// TwinCAT 3 PLC project TE1096_04
// Title: TE1096-04-SISS
// Company: Tegan Innovations Ltd.
// Author: oldschoo1
// ProjectVersion: 1.0.0
// Description: Stopper Insertion/Screw Station, 4th station of the EAGLE production line
// ProgramVersion: 3.1.4024.0
// libraries:
//   Tc2_EthernetIP, * (Beckhoff Automation GmbH)
//   Tc2_MC2, * (Beckhoff Automation GmbH)
//   Tc2_Standard, * (Beckhoff Automation GmbH)
//   Tc2_System, * (Beckhoff Automation GmbH)
//   Tc2_Utilities, * (Beckhoff Automation GmbH)
//   Tc3_Module, * (Beckhoff Automation GmbH)
// project tree:
//   DUTs/00_HMI/ ST_Chart.TcDUT, StPoint.TcDUT, ST_UserLogHMI.TcDUT
//   DUTs/01_MASTER/ E_MachineState.TcDUT, ST_ActiveEventsHMI.TcDUT, ST_AlarmHistory.TcDUT, ST_Events.TcDUT, ST_MachineStatus.TcDUT, ST_MasterCTRL.TcDUT, ST_ModuleCMD.TcDUT, ST_ModuleStatus.TcDUT, ST_SafetyPLC.TcDUT
//   DUTs/02_Y_AXIS/ E_AxisErrorID.TcDUT, E_AxisState.TcDUT, ST_Y_Axis.TcDUT
//   DUTs/03_KISTLER/ E_KistlerErrorID.TcDUT, E_KistlerState.TcDUT, ST_Kistler.TcDUT, ST_KistlerData_Temporary.TcDUT, ST_KistlerData_CMD.TcDUT, ST_KistlerData_Status.TcDUT
//   DUTs/04_SMAC/ E_SmacState.TcDUT, ST_Smac.TcDUT
//   DUTs/04_SMAC/FUNCTIONS/ ST_CYC_MAN.TcDUT, ST_Phasing_Home.TcDUT
//   DUTs/04_SMAC/I_O/ ST_SMAC_I_O.TcDUT
//   DUTs/05_ProcessCycle/ E_ProcessCycle.TcDUT, ST_ProcessReport.TcDUT
//   GVLs/ ETHIP.TcGVL, GVL_CONSTANTS.TcGVL, GVL_MODULES.TcGVL, GVL_PERSISTENT.TcGVL, GVL_HMI.TcGVL, GVL_IO.TcGVL, GVL_MASTER.TcGVL, GVL_UTILITIES.TcGVL
//   / PlcTask.TcTTO, PulseTask.TcTTO
//   POUs/00_MASTER/ D_FaultHandling.TcPOU, PRG_MasterSystemTime.TcPOU, A_Master.TcPOU, B_Safety.TcPOU, C_Machine_CTRL.TcPOU
//   POUs/01_MODULES/AXIS_Y/ PRG_Fault_Axis_Y.TcPOU, Y_Master_Y_Axis.TcPOU
//   POUs/01_MODULES/KISTLER/ K_Master_Kistler.TcPOU, PRG_Fault_Kistler.TcPOU
//   POUs/01_MODULES/SMAC/ PRG_Fault_SMAC.TcPOU, S_Master_SMAC.TcPOU
//   POUs/02_HMI/ A_HMI.TcPOU
//   POUs/03_Utilities/ FB_ArrayOfByte2Real.TcPOU, FB_BytesToReal.TcPOU, FB_Byte_To_Bits.TcPOU, FB_Chart.TcPOU, FB_DistanceMonitor.TcPOU, FB_EventLog.TcPOU, FB_ForceMonitor.TcPOU, FB_GripperCtrl.TcPOU, FB_Real2ArrayOfByte.TcPOU, FB_Scale.TcPOU, FB_TerminalInfo.TcPOU, FB_TimeControl.TcPOU, FUN_PackBoolArrayToByte.TcPOU, FB_UnpackByteToBoolArray.TcPOU, PRG_SysTime.TcPOU, FB_Pulse.TcPOU, PRG_SysPulses.TcPOU
//   POUs/03_Utilities/SMAC/ FB_ErrorReset.TcPOU, FB_SmacCycleMan.TcPOU, FB_SmacInitialization.TcPOU
//   POUs/ MAIN.TcPOU
// real-time tasks:
//   TASK PulseTask: cycle T#2ms, priority 5, ADS port 352
//   TASK PlcTask: cycle T#10ms, priority 20, ADS port 350
// motion (NC):
//   TASK NC-Task 1 SAF: cycle T#2ms, priority 4, ADS port 501
//   TASK NC-Task 1 SVB: cycle T#10ms, priority 8, ADS port 511
//   AXIS Y_Axis (id 1)
//     Dynamic: Acceleration=1231.5, Deceleration=1231.5, Jerk=3694.5
//     Velo: RefSearch=8.21, RefSync=8.21, SlowManual=41.05, FastManual=246.3, Fast=821, Maximum=821
//     MotionControl: Time=1
//     OtherSettings: AllowMotionCmdToSlave=true, DataPersistence=true
//     encoder EncType=19
//       EncPara: ScaleFactorNumerator=10, ScaleFactorDenominator=1048576, MaxCount=#xffffffff
//         SoftEndMinControl: Enable=true, Range=4.3
//         SoftEndMaxControl: Enable=true, Range=111
//     drive DrvType=16
//       DrvPara: MaxCount=#xffffffff, DriveControlDWord=#x00020000
//         Analog: VeloReferenz=903.1, VeloScale=32, TorqueSetpointScale=10, ScaleFactorActTorque=0.1
//         TimeComp: TaskDelayCycles=1
//     controller CtrType=1
//       CtrPara: PriorControlFactor=1
//         PosDiffControl: Range=1.3, Time=0.5
//         Observer: BandWidth=20
// I/O:
//   DEVICE EtherCAT Master (disabled), AmsNetId 192.168.0.127.2.1
//     Term 1 (EK1100) [EK1100 EtherCAT Coupler (2A E-Bus)]
//       Term 2 (EL6070-0033) [EL6070-0033 1Ch. Licence key terminal, individual licences]
//       Term 3 (EL6910) [EL6910, TwinSAFE PLC]
//       Term 4 (EL1918) [EL1918, 8Ch. Safety Input 24V, TwinSAFE]
//         modules: Module 1 (FSOE), Module 2 (FSLOGIC)
//       Term 5 (EL1918) [EL1918, 8Ch. Safety Input 24V, TwinSAFE]
//         modules: Module 1 (FSOE), Module 2 (FSLOGIC)
//       Term 6 (EL2904) [EL2904, 4 Ch. Safety Output 24V, 0.5A, TwinSAFE]
//         modules: Module 1 (FSOES), Module 2 (DO)
//       Term 7 (EL2904) [EL2904, 4 Ch. Safety Output 24V, 0.5A, TwinSAFE]
//         modules: Module 1 (FSOES), Module 2 (DO)
//       Term 8 (EL1809) [EL1809 16Ch. Dig. Input 24V, 3ms]
//       Term 9 (EL1809) [EL1809 16Ch. Dig. Input 24V, 3ms]
//       Term 10 (EL2809-0015) [EL2809-0015 16Ch. Dig. Output 24V DC, 0.35A, not short-circuit proof]
//       Term 11 (EL9576) [EL9576 Brake chopper terminal]
//       Term 12 (EL7211-0010) [EL7211-0010 1Ch. MDP742 Servo motor output stage with OCT (50V, 4.5A RMS)]
//       Term 14 (EL9011) [EL9011 End Terminal]
//     Box 13 (maXYmos) [5877A5847A]
//   DEVICE Device 2 (TC3 EIP Scanner), AmsNetId 192.168.0.127.3.1
//     VLC-2-EIP // <INFO> 192.168.7.180, VLC-2-EIP (ProdCode: 58072, Rev: 2.94, Mac: 00:03:19:45:01:01) </INFO> <EDS> C:\TwinCAT\3.1\Config\Io\EtherNetIP\VLC-2-EIP.eds </EDS>
// variable links:
//   NC-Task 1 SAF/Axes/Y_Axis <-> EtherCAT Master/Term 1 (EK1100)/Term 12 (EL7211-0010)
//     Drive/Inputs/In/nDcOutputTime <-> InfoData/DcOutputShift
//     Drive/Inputs/In/nState1 <-> DRV Statusword/Statusword
//     Drive/Inputs/In/nState2 <-> DRV Statusword/Statusword @bit 8
//     Drive/Inputs/In/nState4 @bit 1 <-> WcState/InputToggle
//     Drive/Inputs/In/nState4 <-> WcState/WcState
//     Drive/Outputs/Out/nCtrl1 <-> DRV Controlword/Controlword
//     Drive/Outputs/Out/nCtrl2 <-> DRV Controlword/Controlword @bit 8
//     Drive/Outputs/Out/nDataOut2 <-> DRV Target velocity/Target velocity
//     Enc/Inputs/In/nDataIn1 <-> FB Position/Position
//     Enc/Inputs/In/nDcInputTime <-> InfoData/DcInputShift
//     Enc/Inputs/In/nState4 @bit 1 <-> WcState/InputToggle
//     Enc/Inputs/In/nState4 <-> WcState/WcState
//   TE1096-04/TE1096-04 Instance <-> Device 2 (TC3 EIP Scanner)/VLC-2-EIP
//     PlcTask Inputs/GVL_MODULES.stSmacIO.inCurrentMacro <-> Connection 1 (Input/Output)/Inputs/I_MacroCallIndicator
//     PlcTask Inputs/GVL_MODULES.stSmacIO.inCurrentPositionLinear <-> Connection 1 (Input/Output)/Inputs/I_PositionActualVal_1
//     PlcTask Inputs/GVL_MODULES.stSmacIO.inCurrentPositionRotative <-> Connection 1 (Input/Output)/Inputs/I_PositionActualVal_2
//     PlcTask Inputs/GVL_MODULES.stSmacIO.inCurrentValueLinear <-> Connection 1 (Input/Output)/Inputs/I_CurrentVal_1
//     PlcTask Inputs/GVL_MODULES.stSmacIO.inCurrentValueRotative <-> Connection 1 (Input/Output)/Inputs/I_CurrentVal_2
//     PlcTask Inputs/GVL_MODULES.stSmacIO.inErrorIDLinear <-> Connection 1 (Input/Output)/Inputs/I_FollowingError_1
//     PlcTask Inputs/GVL_MODULES.stSmacIO.inErrorIDRotative <-> Connection 1 (Input/Output)/Inputs/I_FollowingError_2
//     PlcTask Inputs/GVL_MODULES.stSmacIO.inModeOfOperationLinear <-> Connection 1 (Input/Output)/Inputs/I_ModeofOperationDisplay_1
//     PlcTask Inputs/GVL_MODULES.stSmacIO.inModeOfOperationRotative <-> Connection 1 (Input/Output)/Inputs/I_ModeofOperationDisplay_2
//     PlcTask Inputs/GVL_MODULES.stSmacIO.inStatusWordLinear <-> Connection 1 (Input/Output)/Inputs/I_StatusWord_1
//     PlcTask Inputs/GVL_MODULES.stSmacIO.inStatusWordRotative <-> Connection 1 (Input/Output)/Inputs/I_StatusWord_2
//     PlcTask Outputs/GVL_MODULES.stSmacIO.qnControlWordLinear <-> Connection 1 (Input/Output)/Outputs/O_ControlWord_1
//     PlcTask Outputs/GVL_MODULES.stSmacIO.qnControlWordRotative <-> Connection 1 (Input/Output)/Outputs/O_ControlWord_2
//     PlcTask Outputs/GVL_MODULES.stSmacIO.qnModeOfOperationLinear <-> Connection 1 (Input/Output)/Outputs/O_ModesofOperation_1
//     PlcTask Outputs/GVL_MODULES.stSmacIO.qnModeOfOperationRotative <-> Connection 1 (Input/Output)/Outputs/O_ModesofOperation_2
//     PlcTask Outputs/GVL_MODULES.stSmacIO.qnSetAcceleraionLinear <-> Connection 1 (Input/Output)/Outputs/O_ProfileAcceleration_1
//     PlcTask Outputs/GVL_MODULES.stSmacIO.qnSetAcceleraionRotative <-> Connection 1 (Input/Output)/Outputs/O_ProfileAcceleration_2
//     PlcTask Outputs/GVL_MODULES.stSmacIO.qnSetMacroNumber <-> Connection 1 (Input/Output)/Outputs/O_MacroNumber
//     PlcTask Outputs/GVL_MODULES.stSmacIO.qnSetMaxiumTorqueLinear <-> Connection 1 (Input/Output)/Outputs/O_MaximumTorque_1
//     PlcTask Outputs/GVL_MODULES.stSmacIO.qnSetMaxiumTorqueRotative <-> Connection 1 (Input/Output)/Outputs/O_MaximumTorque_2
//     PlcTask Outputs/GVL_MODULES.stSmacIO.qnSetPointLinear <-> Connection 1 (Input/Output)/Outputs/O_Setpoint_1
//     PlcTask Outputs/GVL_MODULES.stSmacIO.qnSetPointRotative <-> Connection 1 (Input/Output)/Outputs/O_Setpoint_2
//     PlcTask Outputs/GVL_MODULES.stSmacIO.qnSetVelocityLinear <-> Connection 1 (Input/Output)/Outputs/O_ProfileVelocity_1
//     PlcTask Outputs/GVL_MODULES.stSmacIO.qnSetVelocityRotative <-> Connection 1 (Input/Output)/Outputs/O_ProfileVelocity_2
//   TE1096-04/TE1096-04 Instance <-> EtherCAT Master/Box 13 (maXYmos)
//     PlcTask Inputs/GVL_IO.iStatusBytes <-> Inputs0/1 Byte In (0)
//     PlcTask Inputs/GVL_IO.iStatusBytes @bit {8..1592 step 8} <-> Inputs0/1 Byte In ({1..199})  (199 links)
//     PlcTask Inputs/GVL_IO.nKistlermaXYmosState <-> InfoData/State
//     PlcTask Outputs/GVL_IO.qControlBytes <-> Outputs0/1 Byte Out (0)
//     PlcTask Outputs/GVL_IO.qControlBytes @bit {8..1592 step 8} <-> Outputs0/1 Byte Out ({1..199})  (199 links)
//   TE1096-04/TE1096-04 Instance <-> EtherCAT Master/Term 1 (EK1100)
//     PlcTask Inputs/GVL_IO.nEK1100State <-> InfoData/State
//   TE1096-04/TE1096-04 Instance <-> EtherCAT Master/Term 1 (EK1100)/Term 10 (EL2809-0015)
//     PlcTask Inputs/GVL_IO.nEL2809State <-> InfoData/State
//     PlcTask Outputs/GVL_IO.qCycleIndicator_GreenLED <-> Channel 8/Output
//     PlcTask Outputs/GVL_IO.qCycleIndicator_RedLED <-> Channel 7/Output
//     PlcTask Outputs/GVL_IO.qGripperA_Close <-> Channel 3/Output
//     PlcTask Outputs/GVL_IO.qGripperA_Open <-> Channel 4/Output
//     PlcTask Outputs/GVL_IO.qGripperB_Close <-> Channel 5/Output
//     PlcTask Outputs/GVL_IO.qGripperB_Open <-> Channel 6/Output
//     PlcTask Outputs/GVL_IO.qKistlerCTRL_Sig{1..4} <-> Channel {9..12}/Output  (4 links)
//     PlcTask Outputs/GVL_IO.qResetButton_LED <-> Channel 2/Output
//     PlcTask Outputs/GVL_IO.qSmacCTRL_Sig1 <-> Channel 13/Output
//     PlcTask Outputs/GVL_IO.qSmacCTRL_Sig2 <-> Channel 14/Output
//     PlcTask Outputs/GVL_IO.qSmacCTRL_Sig3 <-> Channel 15/Output
//     PlcTask Outputs/GVL_IO.qStartButton_LED <-> Channel 1/Output
//   TE1096-04/TE1096-04 Instance <-> EtherCAT Master/Term 1 (EK1100)/Term 11 (EL9576)
//     PlcTask Inputs/GVL_IO.nEL9576State <-> InfoData/State
//   TE1096-04/TE1096-04 Instance <-> EtherCAT Master/Term 1 (EK1100)/Term 12 (EL7211-0010)
//     PlcTask Inputs/GVL_IO.nEL7211State <-> InfoData/State
//   TE1096-04/TE1096-04 Instance <-> EtherCAT Master/Term 1 (EK1100)/Term 2 (EL6070-0033)
//     PlcTask Inputs/GVL_IO.nEL6070State <-> InfoData/State
//   TE1096-04/TE1096-04 Instance <-> EtherCAT Master/Term 1 (EK1100)/Term 3 (EL6910)
//     PlcTask Inputs/GVL_IO.isDoorClosed <-> StandardInputs/Standard Out Var 21
//     PlcTask Inputs/GVL_IO.isDoorLocked <-> StandardInputs/Standard Out Var 23
//     PlcTask Inputs/GVL_IO.isEStop_OK <-> StandardInputs/Standard Out Var 20
//     PlcTask Inputs/GVL_IO.isLightBeam_NotCrossed <-> StandardInputs/Standard Out Var 25
//     PlcTask Inputs/GVL_IO.isLightBeam_OK <-> StandardInputs/Standard Out Var 26
//     PlcTask Inputs/GVL_IO.isSafetyCom_Error <-> StandardInputs/Standard Out Var 19
//     PlcTask Inputs/GVL_IO.isSafetyFB_Error <-> StandardInputs/Standard Out Var 18
//     PlcTask Inputs/GVL_IO.isSafetyRunning <-> StandardInputs/Standard Out Var 17
//     PlcTask Inputs/GVL_IO.isSafety_OK <-> StandardInputs/Standard Out Var 30
//     PlcTask Inputs/GVL_IO.isTwoHands_SIGNAL <-> StandardInputs/Standard Out Var 28
//     PlcTask Inputs/GVL_IO.nEL6910State <-> InfoData/State
//     PlcTask Outputs/GVL_IO.qsLightBeam_MutingActive <-> StandardOutputs/Standard In Var 24
//     PlcTask Outputs/GVL_IO.qsLockDoorCMD <-> StandardOutputs/Standard In Var 22
//     PlcTask Outputs/GVL_IO.qsSafetyErrorAck <-> StandardOutputs/Standard In Var 1
//     PlcTask Outputs/GVL_IO.qsSafetyRun <-> StandardOutputs/Standard In Var 3
//     PlcTask Outputs/GVL_IO.qsTwoHandsMonitoring <-> StandardOutputs/Standard In Var 27
//   TE1096-04/TE1096-04 Instance <-> EtherCAT Master/Term 1 (EK1100)/Term 4 (EL1918)
//     PlcTask Inputs/GVL_IO.iDoorInterlock_Ch1 <-> Module 1 (FSOE)/FSoE Inputs/FSOE/FSIN Module 4.Input
//     PlcTask Inputs/GVL_IO.iDoorInterlock_Ch2 <-> Module 1 (FSOE)/FSoE Inputs/FSOE/FSIN Module 5.Input
//     PlcTask Inputs/GVL_IO.iDoorInterlock_FB <-> Module 1 (FSOE)/FSoE Inputs/FSOE/FSIN Module 6.Input
//     PlcTask Inputs/GVL_IO.iE_Stop_Ch1 <-> Module 1 (FSOE)/FSoE Inputs/FSOE/FSIN Module 1.Input
//     PlcTask Inputs/GVL_IO.iE_Stop_Ch2 <-> Module 1 (FSOE)/FSoE Inputs/FSOE/FSIN Module 2.Input
//     PlcTask Inputs/GVL_IO.iIndraDrive_Contactor_FB <-> Module 1 (FSOE)/FSoE Inputs/FSOE/FSIN Module 7.Input
//     PlcTask Inputs/GVL_IO.iResetButton <-> Module 1 (FSOE)/FSoE Inputs/FSOE/FSIN Module 3.Input
//     PlcTask Inputs/GVL_IO.iSmacSTO_FB <-> Module 1 (FSOE)/FSoE Inputs/FSOE/FSIN Module 8.Input
//     PlcTask Inputs/GVL_IO.nEL1918_1State <-> InfoData/State
//   TE1096-04/TE1096-04 Instance <-> EtherCAT Master/Term 1 (EK1100)/Term 5 (EL1918)
//     PlcTask Inputs/GVL_IO.iAxis_1_SafetyRelayFB <-> Module 1 (FSOE)/FSoE Inputs/FSOE/FSIN Module 6.Input
//     PlcTask Inputs/GVL_IO.iPilz2_FB <-> Module 1 (FSOE)/FSoE Inputs/FSOE/FSIN Module 5.Input
//     PlcTask Inputs/GVL_IO.iSafetyBeam_Signal <-> Module 1 (FSOE)/FSoE Inputs/FSOE/FSIN Module 7.Input
//     PlcTask Inputs/GVL_IO.iTouchBtn_1_NC <-> Module 1 (FSOE)/FSoE Inputs/FSOE/FSIN Module 1.Input
//     PlcTask Inputs/GVL_IO.iTouchBtn_2_NC <-> Module 1 (FSOE)/FSoE Inputs/FSOE/FSIN Module 2.Input
//     PlcTask Inputs/GVL_IO.iTouchBtn_1_NO <-> Module 1 (FSOE)/FSoE Inputs/FSOE/FSIN Module 3.Input
//     PlcTask Inputs/GVL_IO.iTouchBtn_2_NO <-> Module 1 (FSOE)/FSoE Inputs/FSOE/FSIN Module 4.Input
//     PlcTask Inputs/GVL_IO.nEL1918_2State <-> InfoData/State
//   TE1096-04/TE1096-04 Instance <-> EtherCAT Master/Term 1 (EK1100)/Term 6 (EL2904)
//     PlcTask Inputs/GVL_IO.nEL2904_1State <-> InfoData/State
//   TE1096-04/TE1096-04 Instance <-> EtherCAT Master/Term 1 (EK1100)/Term 7 (EL2904)
//     PlcTask Inputs/GVL_IO.nEL2904_2State <-> InfoData/State
//   TE1096-04/TE1096-04 Instance <-> EtherCAT Master/Term 1 (EK1100)/Term 8 (EL1809)
//     PlcTask Inputs/GVL_IO.iKistlerCTRL_FB1 <-> Channel 9/Input
//     PlcTask Inputs/GVL_IO.iKistlerCTRL_FB2 <-> Channel 10/Input
//     PlcTask Inputs/GVL_IO.iKistlerCTRL_FB3 <-> Channel 11/Input
//     PlcTask Inputs/GVL_IO.iPSU_1_OK <-> Channel 3/Input
//     PlcTask Inputs/GVL_IO.iPSU_2_OK <-> Channel 4/Input
//     PlcTask Inputs/GVL_IO.iPSU_3_OK <-> Channel 5/Input
//     PlcTask Inputs/GVL_IO.iSmacCTRL_FB1 <-> Channel 13/Input
//     PlcTask Inputs/GVL_IO.iSmacCTRL_FB2 <-> Channel 14/Input
//     PlcTask Inputs/GVL_IO.iSmacCTRL_FB3 <-> Channel 15/Input
//     PlcTask Inputs/GVL_IO.iStartButton <-> Channel 1/Input
//     PlcTask Inputs/GVL_IO.iStopButton <-> Channel 2/Input
//     PlcTask Inputs/GVL_IO.nEL1809_1State <-> InfoData/State
//   TE1096-04/TE1096-04 Instance <-> EtherCAT Master/Term 1 (EK1100)/Term 9 (EL1809)
//     PlcTask Inputs/GVL_IO.iGripperA_ClosedSensor <-> Channel 4/Input
//     PlcTask Inputs/GVL_IO.iGripperB_ClosedSensor <-> Channel 5/Input
//     PlcTask Inputs/GVL_IO.iPartA_PresentSensor <-> Channel 2/Input
//     PlcTask Inputs/GVL_IO.iPartB_PresentSensor <-> Channel 3/Input
//     PlcTask Inputs/GVL_IO.iPuck_PresentSensor <-> Channel 1/Input
//     PlcTask Inputs/GVL_IO.nEL1809_2State <-> InfoData/State
//   TE1096-04/TE1096-04 Instance <-> NC-Task 1 SAF/Axes/Y_Axis
//     PlcTask Inputs/Y_Master_Y_Axis.refY_Axis.NcToPlc <-> Outputs/ToPlc
//     PlcTask Outputs/Y_Master_Y_Axis.refY_Axis.PlcToNc <-> Inputs/FromPlc
//   (this object) <-> EtherCAT Master
//     Term 1 (EK1100)/Term 3 (EL6910)/ConnectionInputs/Message_13 TxPDO <-> Term 1 (EK1100)/Term 4 (EL1918)/Module 1 (FSOE)/FSoE Outputs/FSOE
//     Term 1 (EK1100)/Term 3 (EL6910)/ConnectionInputs/Message_14 TxPDO <-> Term 1 (EK1100)/Term 5 (EL1918)/Module 1 (FSOE)/FSoE Outputs/FSOE
//     Term 1 (EK1100)/Term 3 (EL6910)/ConnectionInputs/Message_15 TxPDO <-> Term 1 (EK1100)/Term 6 (EL2904)/Module 1 (FSOES)/RxPDO/FSOE
//     Term 1 (EK1100)/Term 3 (EL6910)/ConnectionInputs/Message_16 TxPDO <-> Term 1 (EK1100)/Term 7 (EL2904)/Module 1 (FSOES)/RxPDO/FSOE
//     Term 1 (EK1100)/Term 3 (EL6910)/ConnectionOutputs/Message_13 RxPDO <-> Term 1 (EK1100)/Term 4 (EL1918)/Module 1 (FSOE)/FSoE Inputs/FSOE
//     Term 1 (EK1100)/Term 3 (EL6910)/ConnectionOutputs/Message_14 RxPDO <-> Term 1 (EK1100)/Term 5 (EL1918)/Module 1 (FSOE)/FSoE Inputs/FSOE
//     Term 1 (EK1100)/Term 3 (EL6910)/ConnectionOutputs/Message_15 RxPDO <-> Term 1 (EK1100)/Term 6 (EL2904)/Module 1 (FSOES)/TxPDO/FSOE
//     Term 1 (EK1100)/Term 3 (EL6910)/ConnectionOutputs/Message_16 RxPDO <-> Term 1 (EK1100)/Term 7 (EL2904)/Module 1 (FSOES)/TxPDO/FSOE
//     Term 1 (EK1100)/Term 4 (EL1918)/Module 1 (FSOE)/FSoE Inputs/FSOE <-> Term 1 (EK1100)/Term 3 (EL6910)/ConnectionOutputs/Message_13 RxPDO
//     Term 1 (EK1100)/Term 5 (EL1918)/Module 1 (FSOE)/FSoE Inputs/FSOE <-> Term 1 (EK1100)/Term 3 (EL6910)/ConnectionOutputs/Message_14 RxPDO
//     Term 1 (EK1100)/Term 4 (EL1918)/Module 1 (FSOE)/FSoE Outputs/FSOE <-> Term 1 (EK1100)/Term 3 (EL6910)/ConnectionInputs/Message_13 TxPDO
//     Term 1 (EK1100)/Term 5 (EL1918)/Module 1 (FSOE)/FSoE Outputs/FSOE <-> Term 1 (EK1100)/Term 3 (EL6910)/ConnectionInputs/Message_14 TxPDO
//     Term 1 (EK1100)/Term 6 (EL2904)/Module 1 (FSOES)/RxPDO/FSOE <-> Term 1 (EK1100)/Term 3 (EL6910)/ConnectionInputs/Message_15 TxPDO
//     Term 1 (EK1100)/Term 7 (EL2904)/Module 1 (FSOES)/RxPDO/FSOE <-> Term 1 (EK1100)/Term 3 (EL6910)/ConnectionInputs/Message_16 TxPDO
//     Term 1 (EK1100)/Term 6 (EL2904)/Module 1 (FSOES)/TxPDO/FSOE <-> Term 1 (EK1100)/Term 3 (EL6910)/ConnectionOutputs/Message_15 RxPDO
//     Term 1 (EK1100)/Term 7 (EL2904)/Module 1 (FSOES)/TxPDO/FSOE <-> Term 1 (EK1100)/Term 3 (EL6910)/ConnectionOutputs/Message_16 RxPDO

CONFIGURATION TE1096_04
    RESOURCE PLC ON TwinCAT3
        TASK PlcTask(INTERVAL := T#10ms, PRIORITY := 20);
        TASK PulseTask(INTERVAL := T#2ms, PRIORITY := 5);
        PROGRAM MAIN WITH PlcTask : MAIN;
        PROGRAM PRG_SysPulses WITH PulseTask : PRG_SysPulses;
    END_RESOURCE
END_CONFIGURATION

// ---- DUTs/00_HMI/ST_Chart.TcDUT
TYPE ST_Chart :
STRUCT
        Distance : REAL;
        Force    : REAL;
END_STRUCT
END_TYPE

// ---- DUTs/00_HMI/StPoint.TcDUT
TYPE StPoint :
STRUCT
    x : REAL;
    y : REAL;
END_STRUCT
END_TYPE

// ---- DUTs/00_HMI/ST_UserLogHMI.TcDUT
TYPE ST_UserLogHMI :
STRUCT
	UserLog					: T_MaxSTring;
	UserLogTime				: STRING;
	UserLogDate				: STRING;
END_STRUCT
END_TYPE

// ---- DUTs/01_MASTER/E_MachineState.TcDUT
{attribute 'qualified_only'}
{attribute 'strict'}
TYPE E_MachineState :
( // Enum: State of the m/c
	
	SYSTEM_POWER_UP			:=0,
	IMMEDIATE_STOPPED		:=100,
	SYSTEM_INITIALISING		:=110,
	SYSTEM_READY_TO_START	:=120,
	SYSTEM_AUTO_CYCLE		:=130,
	SYSTEM_STANDBY			:=140,
	STOPPING				:=150,
	CYCLE_STOPPED			:=160,
	MANUAL_MODE				:=170,
	IMMEDIATE_FAULT			:=190,
	CYCLE_STOP_FAULT		:=200
	
	//-----------------------------------------------------------------------------------------------------------------------oldschoo1
);
END_TYPE

// ---- DUTs/01_MASTER/ST_ActiveEventsHMI.TcDUT
TYPE ST_ActiveEventsHMI :
STRUCT
	sActiveEvents					: T_MaxSTring;
END_STRUCT
END_TYPE

// ---- DUTs/01_MASTER/ST_AlarmHistory.TcDUT
TYPE ST_AlarmHistory :
STRUCT
	
	sEventlog 	:T_MaxSTring;
	sDate		:T_MaxSTring;
	sTime		:T_MaxSTring;
END_STRUCT
END_TYPE

// ---- DUTs/01_MASTER/ST_Events.TcDUT
TYPE ST_Events :
STRUCT
	bImmediateFault				:BOOL;
	bCycleStopFault				:BOOL;
	bCycleStopRequest			:BOOL;

	bEventTextsSet				:BOOL; //True after event texts are set 
	aEventFlags					:ARRAY[0..127] OF BOOL;
	aEventTimers				:ARRAY[0..127] OF TON;
	aEventTexts					:ARRAY[0..127] OF T_MaxString;
END_STRUCT
END_TYPE

// ---- DUTs/01_MASTER/ST_MachineStatus.TcDUT
TYPE ST_MachineStatus :
STRUCT
// Struct: Machine Status
	
	eMachineState				:E_MachineState;
	stMasterCTRL				:ST_MasterCTRL;
	
	// Status Flags:
	bSystemPowerUp 				:BOOL;
	bImmediateStopped 			:BOOL;
	bInitialising 				:BOOL;
	bReadyToStart 				:BOOL;
	bAutoCycle 					:BOOL;
	bStandby 					:BOOL;
	bStopping					:BOOL;	
	bCycleStopped 				:BOOL;
	bImmediateFault 			:BOOL;
	bCycleStopFault 			:BOOL;
	bManualMode					:BOOL;
	bProcessCycle				:BOOL;	// True when Operation in Progress
	
	// HMI data
	sMachineStatusText			:STRING;
	nMachineStatusTxtCol		:DWORD;
	nMachineStatusColour		:DWORD;
	sBannerTextColor			:STRING;
	sBannerBckColor				:STRING;	

	
	//-----------------------------------------------------------------------------------------------------------------------oldschoo1
	
END_STRUCT
END_TYPE

// ---- DUTs/01_MASTER/ST_MasterCTRL.TcDUT
TYPE ST_MasterCTRL :
STRUCT
	

	// Request Flags
	bHoming_Request						:BOOL;
	bProccess_Request					:BOOL;
	bStop_Request						:BOOL;
	bAbortAction_Request				:BOOL;
	bManualModeRequest					:BOOL;
	
	bCycleStopRequest					:BOOL;		
	bAllActionsStopped					:BOOL;
	bCycleStopFault						:BOOL;
	bNoMachineImmediateFault			:BOOL;
	bNoCycleStopFault					:BOOL;	
	bAllModulesReady					:BOOL;

	// Feedback Flags
	bAllModules_Homed					:BOOL;
	bAllModules_Stopped					:BOOL;
	bAllModules_Aborted					:BOOL;
	bPowerUpTimerComplete				:BOOL;

	
//-------------------------------------------------------------------------------oldschoo1
		
END_STRUCT
END_TYPE

// ---- DUTs/01_MASTER/ST_ModuleCMD.TcDUT
TYPE ST_ModuleCMD :
STRUCT
//Universal Module CMD Struct

    bEnable       			:BOOL;	// Request module to activate devices
	bExecute				:BOOL;	// Request module to execute CMD
    bReset        			:BOOL;	// Request module to reset error or state
    bAbort        			:BOOL;	// Emergency stop or cancel current task
	
	nTaskID       			:UINT;	// Request a Task by its ID	
    nTargetState  			:UINT;	// State-machine target request
    bManualMode   			:BOOL;	// Request Manual Mode(jog mode)
	
	bSetAction_1     		:REAL;	// Set Action
	bSetAction_2     		:REAL;	// Set Action 
	bSetAction_3     		:REAL;	// Set Action
	bSetAction_4     		:REAL;	// Set Action
	    
    rSetpoint_1     		:REAL;	// Setpoint value
	rSetpoint_2     		:REAL;	// Setpoint value 
	rSetpoint_3     		:REAL;	// Setpoint value 
	rSetpoint_4     		:REAL;	// Setpoint value 
	
	bFixtureGripper			:BOOL;
	bGuideGripper			:BOOL;
	
	
//-----------------------------------------------------------------------------oldschoo1


END_STRUCT
END_TYPE

// ---- DUTs/01_MASTER/ST_ModuleStatus.TcDUT
TYPE ST_ModuleStatus :
STRUCT
//Universal Module STATUS Struct

	bReady        			:BOOL;	// Module initialized and ready for CMD
    bBusy         			:BOOL;	// Module is busy processing a request
    bDone         			:BOOL;	// Operation successfully completed
    bError        			:BOOL;	// Error occurred
    nErrorID      			:INT;	// Error code (ideally enum-based)
	
	bActionInProggress		:BOOL;	// Device is Busy doing the Job
    
    bInPosition_1   		:BOOL;	// Module has reached target Setpoint_1
	bInPosition_2   		:BOOL;	// Module has reached target Setpoint_2
	bInPosition_3   		:BOOL;	// Module has reached target Setpoint_3
	bInPosition_4   		:BOOL;	// Module has reached target Setpoint_4
	
	nCurrentTaskID			:UINT;	// Current Task ID
    nCurrentState 			:UINT;	// Current State
	
	bFirstPartOfCycleDone	:BOOL; //SMAC

	

//-----------------------------------------------------------------------------------------oldschoo1	


END_STRUCT
END_TYPE

// ---- DUTs/01_MASTER/ST_SafetyPLC.TcDUT
TYPE ST_SafetyPLC :
STRUCT
// Struct: Safety PLC
	

	// Safety CMDs	
	bRunSafety                          :BOOL;  // Start Safety CMD
	bAckSafetyError						:BOOL;	// Safety Error Acknowledge

	bTwoHands_MonitorCMD  	            :BOOL;  // 2Hands needed to trigger Parts Proccessing 
	bLightBeam_MuteCMD					:BOOL;	// SICK Safety LightBeam - Muting active
	bLockDoor_CMD						:BOOL;	// CMD to lock the Door
	
	// Safety Status
	bSafetyRunning                      :BOOL;  // TwinSAFE running
	bSafetyFB_Error	 					:BOOL;	// TwinSAFE modules Feedback Error
	bSafetyCom_Error 					:BOOL;	// TwinSAFE Communication error	
	bSafety_OK							:BOOL;	// All safety gear OK
	
	// Safety Gear
    bEStop_OK	                        :BOOL;  // E-Stop OK
	bEStop_Pressed						:BOOL;	// E-Stop Pressed
	bDoorClosed							:BOOL;	// Door Closed
	bDoorLocked							:BOOL;	// Door Locked
	bDoorOpen							:BOOL;	// Door Open
	bLightBeam_Crossed					:BOOL;	// SICK Safety LightBeam - Crosed!
	bTwoHands_Signal					:BOOL;	// TwoHands - Both Buttons activated

	// Terminal Inputs
	bE_Stop_Ch1							:BOOL;	// E-Stop ch1
	bE_Stop_Ch2							:BOOL;	// E-Stop ch2                               	
	bResetButton						:BOOL;	// Reset Button	
	bDoorInterlock_Ch1					:BOOL;	// Door Closed ch1
	bDoorInterlock_Ch2					:BOOL;	// Door Closed ch2	                                	
	bDoorInterlock_FB					:BOOL;	// Door Feedback Sig.
	bIndraDrive_Contactor_FB			:BOOL;	// Kistler drive Safety Contactor Feedback
	bSmacSTO_FB							:BOOL;	// SMACK Safe Torque OFF Feedback
	bTouchBtn_1_NC						:BOOL;	// Safety Touch Button 1 
	bTouchBtn_2_NC						:BOOL;	// Safety Touch Button 2                               	
	bTouchBtn_1_NO						:BOOL;	// Safety Touch Button 1
	bTouchBtn_2_NO						:BOOL;	// Safety Touch Button 2
	bPilz2_FB							:BOOL;	// Pilz Safety Relay 2 Feedback
	bAxis_1_SafetyRelayFB				:BOOL;	// AXIS 1 Safety Relay Feedback
	
	
	
	nSafetyTerminalStatus				:UINT;	//Ethercat Terminal Status

		//-------------------------------------------------------------------------------oldschoo1
		
END_STRUCT
END_TYPE

// ---- DUTs/02_Y_AXIS/E_AxisErrorID.TcDUT
{attribute 'qualified_only'}
{attribute 'strict'}
TYPE E_AxisErrorID :
(
	NO_ERROR			:=0,
	POWER_UP_ERROR		:=10,
	HOMING_ERROR		:=20,
	MOVEMENT_ERROR		:=30,
	TIMEOUT_ERROR		:=40
	//---------------------o1
);
END_TYPE

// ---- DUTs/02_Y_AXIS/E_AxisState.TcDUT
{attribute 'qualified_only'}
{attribute 'strict'}
TYPE E_AxisState :
(

	ABORTED				:=10,
	ENABLE_POWER		:=20,
	RESET_ERROR			:=30,
	HOMING				:=33,
	AXIS_READY			:=40,
	GET_TARGET			:=50,
	MOVE_ABS			:=60,
	MOVING_ABS			:=70,
	MOVE_REL			:=80,
	MOVING_REL			:=90,
	IN_TARGET_POS		:=100,
	ERROR				:=110,
	MANUAL_MODE			:=120
//------------------------------oldschoo1	
);
END_TYPE

// ---- DUTs/02_Y_AXIS/ST_Y_Axis.TcDUT
TYPE ST_Y_Axis :
STRUCT
	
	// Parameters
	posHome      					:LREAL;					//Home Position
	posWorkPositions   				:ARRAY[1..3] OF LREAL;	//Array of Positions
	fPositionOffsets   				:ARRAY[1..3] OF LREAL;	//Array of Position Offsets

    bSetToHome     					:BOOL;					//Set Position Home
    bSetToPosition    				:ARRAY[1..3] OF BOOL;	//Flags to Request a Position
	
	fTargetVelocity					:LREAL;					//Set Target Velocity
	fRetractVelocity				:LREAL;					//Set Retract Velocity
	
	// Feedback
	bAxis_1_InErrorState			:BOOL;
	nAxis_1_nErrorID				:UINT;
	bAxis_1_SafetyRelayFB			:BOOL;					//Axis Safety Relay Feedback
	
//------------------------------------------------------------------------------------------------oldschoo1


END_STRUCT
END_TYPE

(*
***INFO
posPoints[1]:= 15.00;		//Work position to pick the Screw
posPoints[2]:= 33.00;		//Work position to do Screwing and Pressing 
posPoints[3]:= 100.00;		//Position to take out the Pack Fixture
*)

// ---- DUTs/03_KISTLER/E_KistlerErrorID.TcDUT
{attribute 'qualified_only'}
{attribute 'strict'}
TYPE E_KistlerErrorID :
(
	NO_ERROR				:=0,
	COMUNICATION_ERROR		:=10,
	ENABLE_DRIVE_ERROR		:=20,
	PROCESS_ERROR			:=30,
	ACTION_TIMEOUT_ERROR	:=40
	
	
);
END_TYPE

// ---- DUTs/03_KISTLER/E_KistlerState.TcDUT
{attribute 'qualified_only'}
{attribute 'strict'}
TYPE E_KistlerState :
(
	ABORTED				:=10,
	ENABLE_PLC_CTRL		:=11,
	SELECT_MP			:=12,
	ENABLE_DRIVE		:=20,
	RESET_ERROR			:=30,
	GOTO_HOME_POS		:=33,
	SET_PARAMETERS		:=40,
	PRESS_READY			:=50,
	PRESS_CYCLE			:=60,
	WAIT_CYCLE_DONE		:=70,
	RECORD_CYCLE_DATA	:=80,
	JOG_MODE			:=100,
	ERROR				:=110,
	MANUAL				:=120
	
//------------------------------oldschoo1
);
END_TYPE

// ---- DUTs/03_KISTLER/ST_Kistler.TcDUT
TYPE ST_Kistler :
STRUCT


	// EtherCAT communication
	st_TelegramDataOut                   	:ARRAY[0..199]OF BYTE; 	// Channels/Triggers
	st_TelegramDataIn                  		:ARRAY[0..199]OF BYTE; // Mirror/Statuses

	
	// I/O communication
	bKistlerCTRL_FB1						:BOOL;	// Channel 09 - Kistler CTRL - Feedback Signal 1	
	bKistlerCTRL_FB2						:BOOL;	// Channel 10 - Kistler CTRL - Feedback Signal 2	
	bKistlerCTRL_FB3						:BOOL;	// Channel 11 - Kistler CTRL - Feedback Signal 3

	bKistlerCTRL_Sig1						:BOOL;	// Channel 09 - Kistler CTRL Signal 1
	bKistlerCTRL_Sig2						:BOOL;	// Channel 10 - Kistler CTRL Signal 2
	bKistlerCTRL_Sig3						:BOOL;	// Channel 11 - Kistler CTRL Signal 3
	bKistlerCTRL_Sig4						:BOOL;	// Channel 12 - Kistler CTRL Signal 4
	

//---------------------------------------------------------------------------------------------------oldschoo1
	
END_STRUCT
END_TYPE

// ---- DUTs/03_KISTLER/ST_KistlerData_Temporary.TcDUT
TYPE ST_KistlerData_Temporary :
STRUCT

//CMDs
arrOutBits : ARRAY[0..199]OF ARRAY[0..7]OF BOOL;

//Statuses
arrInBits  : ARRAY[0..199]OF ARRAY[0..7]OF BOOL;

//--------------------------------------oldschoo1

END_STRUCT
END_TYPE

// ---- DUTs/03_KISTLER/ST_KistlerData_CMD.TcDUT
TYPE ST_KistlerData_CMD :
STRUCT	
(*********************************Telegram Data***************************************)	

//Byte 0 - Basic Control CMDs
	  bStart          					:BOOL;	// 0.0 START – pulse to trigger cycle
	  bTareY          					:BOOL;	// 0.1 TARE-Y
	  bZeroX          					:BOOL;	// 0.2 ZERO-X
	  bSTestX        					:BOOL;	// 0.3 S-TEST-X
	  bSTestY        					:BOOL;	// 0.4 S-TEST-Y
	  _r0_5          					:BOOL;	// 0.5 reserved
	  bMasterMeas     					:BOOL;	// 0.6 MASTER-MEAS
	  bIncZero        					:BOOL;	// 0.7 INC-ZERO
	
//Byte 1 - Login 
	  bAckAdminGlobal 					:BOOL;	// 1.0 ACK-ADMIN-GLOBAL
	  bAckAdmin		 					:BOOL;	// 1.1 ACK-ADMIN
	  _r1_2        						:BOOL;	// 1.2 reserved
	  bAccess         					:BOOL;	// 1.3 ACCESS
	  bAuto           					:BOOL;	// 1.4 AUTO
	  bStatReset      					:BOOL;	// 1.5 STAT-RESET
	  bStatDisable    					:BOOL;	// 1.6 STAT-DISABLE
	  bTareExtY       					:BOOL;	// 1.7 TARE-EXTENDED-Y
	
//Byte 2 - Measurement PRG Selection
	  mpNumber        					:ARRAY[0..6]OF BOOL;//MP Number
	  _r2_7           					:BOOL;	// 2.7 reserved
	
//Byte 3 – Reserved
	  _byte3							:BYTE;	// reserved
//Byte 4 – Configurable Input Signals
	  _byte4							:BYTE;	// reserved
//Byte 5 – Reserved
	  _byte5							:BYTE;	// reserved
//Byte 6 – Reserved
	  _byte6							:BYTE;	// reserved
//Byte 7 – Reserved
	  _byte7							:BYTE;	// reserved
//Byte 3 – Reserved
	  _byte8							:BYTE;	// reserved
	
//Byte 9 – Drive/Sequence CMDs
	  bDriveEnable    					:BOOL;	// 9.0 DRIVE-ENABLE
	  bRunSequence    					:BOOL;	// 9.1 RUN-SEQUENCE
	  bDriveToHome    					:BOOL;	// 9.2 DRIVE-TO-HOMEPOS
	  bDriveToRef     					:BOOL;	// 9.3 DRIVE-TO-REFPOS
	  bJogFwd         					:BOOL;	// 9.4 JOG-FW
	  bJogBack        					:BOOL;	// 9.5 JOG-BW
	  bContinueWait   					:BOOL;	// 9.6 CONTINUE-FROM-WAIT
	  bBrakeTest      					:BOOL;	// 9.7 MANUAL-BRAKE-TEST
	
//Byte 10 – Extended Stop Request
	  _r10_0to2       					:ARRAY[0..2]OF BOOL;
	  bSeqExtStopReq  					:BOOL;	// 10.3 SEQ-EXT-STOP-REQ
	  _r10_4to7       					:ARRAY[4..7]OF BOOL;
	
//Byte 11 – Reserved
	  _byte11            				:BYTE;	// reserved
	
//Byte 12 – Current Sequence Flags
	  bCurrSeqMain    					:BOOL;	// 12.0 CURRENT-SEQUENCE-0
	  bCurrSeqSub     					:BOOL;	// 12.1 CURRENT-SEQUENCE-1
	  _r12_2to7       					:ARRAY[2..7]OF BOOL;
	
//Byte 13 – Reserved
	  _byte13            				:BYTE;	// reserved
	
//Byte 14 – Page Control (0…127)
	  pageControl     					:BYTE;	// 14.0…14.6 CFG-MP
	
//Bytes 15…19 – Fieldbus Config Bits
	  _r15            					:BYTE;
	  cfgAddress      					:BYTE;	// 16.0…16.7 CFG-ADDRESS
	  cfgLength       					:BYTE;	// 17.0…17.7 CFG-LENGTH
	  cfgSelectPage   					:BYTE;	// 18.0…18.2 SELECT-PAGE
	  saveToMP_Strobe 					:BYTE;	// 19.0…19.7 SAVE/STROBE etc.
	  
(************************************************************************************)
	
(*************************************Payload****************************************)

//Bytes 20…199 – Free Payload
	  spare           					:ARRAY[20..199]OF BYTE;
	  
//---------------------------------------------------------------------------oldschoo1
END_STRUCT
END_TYPE

// ---- DUTs/03_KISTLER/ST_KistlerData_Status.TcDUT
TYPE ST_KistlerData_Status :
STRUCT
(*********************************Telegram Data***************************************)

//Byte 0 – Mirror Basic Control
      bStart_Mirror          			:BOOL; // 0.0 MIRROR-START
      bTareY_Mirror          			:BOOL; // 0.1 MIRROR-TARE-Y
      bZeroX_Mirror          			:BOOL; // 0.2 MIRROR-ZERO-X
      bSTestX_Mirror         			:BOOL; // 0.3 MIRROR-S-TEST-X
      bSTestY_Mirror         			:BOOL; // 0.4 MIRROR-S-TEST-Y
      _r0_5                  			:BOOL; // 0.5 reserved
      bMasterMeas_Mirror     			:BOOL; // 0.6 MIRROR-MASTER-MEAS
      bIncZero_Mirror        			:BOOL; // 0.7 MIRROR-INC-ZERO
      
//Byte 1 – Mirror Login
      bAckAdminGlobal_Mirror 			:BOOL; // 1.0 MIRROR-ACK-ADMIN-GLOBAL
      bAckAdmin_Mirror       			:BOOL; // 1.1 MIRROR-ACK-ADMIN
      _r1_2                  			:BOOL; // 1.2 reserved
      bAccess_Mirror         			:BOOL; // 1.3 MIRROR-ACCESS
      bAuto_Mirror           			:BOOL; // 1.4 MIRROR-AUTO
      bStatReset_Mirror      			:BOOL; // 1.5 MIRROR-STAT-RESET
      bStatDisable_Mirror    			:BOOL; // 1.6 MIRROR-STAT-DISABLE
      bTareExtY_Mirror       			:BOOL; // 1.7 MIRROR-TARE-EXTENDED-Y
      
//Byte 2 – Mirror MP Selection
      mpNumber_Mirror        			:ARRAY[0..6]OF BOOL; // MP-Number mirrored
      _r2_7                  			:BOOL; // 2.7 reserved
      
//Byte 3 – Service & Brake
      _r3_0to1               			:ARRAY[0..1]OF BOOL;
      bResetSNGen_Mirror     			:BOOL; // 3.2 RESET-SN-GENERATOR (mirror)
      _r3_3to4               			:ARRAY[3..4]OF BOOL;
      bBrakeTestActive       			:BOOL; // 3.5 BRAKETEST-ACTIVE
      bExportPvt_Mirror      			:BOOL; // 3.6 MIRROR-EXPORT-PVT-START
      _r3_7                  			:BOOL; // 3.7 reserved
      
//Byte 4 – Mirror Configurable Inputs
      bIUni_Mirror           			:ARRAY[0..7]OF BOOL; //4.0…4.7 MIRROR-I-UNI-0…7
      
//Byte 5 – Reserved
      _byte5                 			:BYTE; // reserved
      
//Byte 6 – Global Status Flags
      bReady                 			:BOOL; // 6.0 READY
      bOkTotal               			:BOOL; // 6.1 OK-TOTAL
      bNokTotal              			:BOOL; // 6.2 NOK-TOTAL
      bNoPass                			:BOOL; // 6.3 NO-PASS
      _r6_4to5               			:ARRAY[4..5]OF BOOL;
      bWarning               			:BOOL; // 6.6 WARNING
      bAlarm                 			:BOOL; // 6.7 ALARM
	  
	  
//Byte 8 – O_UNI Digital Outputs
	  bO_UNI           					:ARRAY[0..7]OF BOOL;
      
//Byte 7 – Switching / User Signals
      bS1                    			:BOOL; // 7.0 S1
      bS2                    			:BOOL; // 7.1 S2
      _r7_2to7               			:ARRAY[2..7]OF BOOL;
      
//Byte 8 – Universal Outputs
      _byte8                 			:BYTE; // O-UNI (user-configurable) or reserved
      
//Byte 9 – Mirror Drive/Sequence
      bDriveEnable_Mirror    			:BOOL; // 9.0 MIRROR-DRIVE-ENABLE
      bRunSequence_Mirror    			:BOOL; // 9.1 MIRROR-RUN-SEQUENCE
      bDriveHome_Mirror      			:BOOL; // 9.2 MIRROR-DRIVE-TO-HOMEPOS
      bDriveRef_Mirror       			:BOOL; // 9.3 MIRROR-DRIVE-TO-REFPOS
      bJogFwd_Mirror         			:BOOL; // 9.4 MIRROR-JOG-FW
      bJogBack_Mirror        			:BOOL; // 9.5 MIRROR-JOG-BW
      bWaitRequest           			:BOOL; // 9.6 WAIT-REQUEST
      bBrakeTestDone         			:BOOL; // 9.7 BRAKETEST-DONE
      
//Byte 10 – Sequence State
      bSeqStopped            			:BOOL; // 10.0 SEQUENCE-STOPPED
      bSeqEnd                			:BOOL; // 10.1 SEQUENCE-END
      bOnlineEoNok           			:BOOL; // 10.2 ONLINE-EO-NOK
      bSeqExtStop            			:BOOL; // 10.3 EXTERN-STOP
      bSeqError              			:BOOL; // 10.4 SEQUENCE-ERROR
      bDriveEnabled          			:BOOL; // 10.5 DRIVE-ENABLED
      bHomePosReached        			:BOOL; // 10.6 HOMEPOS-REACHED
      bRefPosReached         			:BOOL; // 10.7 REFPOS-REACHED
      
//Byte 11 – Servo & Safety
      bStandstill            			:BOOL; // 11.0 STANDSTILL
      bBrakeTestReq          			:BOOL; // 11.1 BRAKETEST-REQUIRED
      bServoWarn             			:BOOL; // 11.2 SERVO-WARNING
      bServoError            			:BOOL; // 11.3 SERVO-ERROR
      bSMES_Or_STO           			:BOOL; // 11.4 SMES / STO
      bSMST2                 			:BOOL; // 11.5 SMST2 active
      bSMM1                  			:BOOL; // 11.6 SMM1 active
      bUserModeActive        			:BOOL; // 11.7 USER-MODE-ACTIVE
      
//Byte 12 – Mirror Current Sequence
      bCurrSeqMain_Mirror    			:BOOL; // 12.0 MIRROR-CURRENT-SEQUENCE-0
      bCurrSeqSub_Mirror     			:BOOL; // 12.1 MIRROR-CURRENT-SEQUENCE-1
      _r12_2to7              			:ARRAY[2..7]OF BOOL;
      
//Byte 13 – Sequence Label-ID
      seqLabelID             			:BYTE; // 13.0…13.4 LABEL-ID (0…31),Upper bits reserved
      
//Byte 14 – Mirror CFG-MP
      pageControl_Mirror     			:BYTE; // 14.0…14.6 MIRROR-CFG-MP, 14.7 reserved
      
//Byte 15 – Reserved
      _byte15                			:BYTE; // reserved
      
//Byte 16 – Mirror CFG-ADDRESS
      cfgAddress_Mirror      			:BYTE; // 16.0…16.7 MIRROR-CFG-ADDRESS
      
//Byte 17 – Mirror CFG-LENGTH
      cfgLength_Mirror       			:BYTE; // 17.0…17.7 MIRROR-CFG-LENGTH
      
//Byte 18 – Mirror Page Select
      cfgSelectPage_Mirror   			:BYTE; // 18.0…18.2 MIRROR-SELECT-PAGE, Rest reserved
      
//Byte 19 – Device / Transfer Flags
      bTransmissionFault     			:BOOL; // 19.0 TRANSMISSION-FAULT
      bAck                   			:BOOL; // 19.1 ACK
      bDeviceAvailable       			:BOOL; // 19.2 DEVICE-AVAILABLE
      _r19_3                 			:BOOL; // 19.3 reserved
      bMpChanged             			:BOOL; // 19.4 CHANGED-SELECTED-MP
      _r19_5                 			:BOOL; // 19.5 reserved
      bGlobalChanged         			:BOOL; // 19.6 CHANGED-GLOBAL
      bBackupComplete        			:BOOL; // 19.7 BACKUP-COMPLETE
      
(*************************************************************************************)
      
(*************************************Payload*****************************************)

//Bytes 20 … 23  - live X value   (factory name  pvCurrentValueX)
	 pvCurrentValueX                    :ARRAY[20..23]OF BYTE;
	 
//Bytes 24 … 27  - live Y value   (factory name  pvCurrentValueY)
	 pvCurrentValueY                    :ARRAY[24..27]OF BYTE;
	 
//Bytes 28 … 35  - 8-byte Alarm/status field
    statusAlarm     					:ARRAY[28..35]OF BYTE;
	
//Bytes 20…199 – Free Payload
    spare           					:ARRAY[36..199]OF BYTE;
//if u r reading this, then God <3 u  
//---------------------------------------------------------------------------oldschoo1
END_STRUCT
END_TYPE

// ---- DUTs/04_SMAC/E_SmacState.TcDUT
{attribute 'qualified_only'}
{attribute 'strict'}
TYPE E_SmacState :
(
	ABORTED				:=10,
	RESET_ERROR			:=30,
	HOMING				:=33,
	AXIS_READY			:=40,
	Cycle_Pick_Part		:=50,
	Cycle_Screw			:=60,
	ERROR				:=110,
	MANUAL				:=120,
	RECORD_CYCLE_DATA	:=140
);
END_TYPE

// ---- DUTs/04_SMAC/FUNCTIONS/ST_CYC_MAN.TcDUT
TYPE ST_CYC_MAN :
STRUCT
///////////////////////////////////////MANUAL//////////////////////////////////////////////////
		bManual_fbSmacCycleMan 						: BOOL;
//SETTINGS:(REMOVE VALUES ONCE MANUAL MODE IMPLEMENTED)
		
		nLinearVel									: DINT;//	:= 8;//8 mm/s
		nLinearAcc									: DINT;//	:= 58000;//58000 mm2/s
		nLinearSetPoint								: DINT;//	:= 50;//50 mm
		nLinearTorque								: INT;//	:= 13;//14v
	
		nRotativeVel								: DINT;//	:= 77;//77mm
		nRotativeAcc								: DINT;//	:= 58000;//58000mm2/s
		nRotativeSetPoint							: DINT;//	:= -22000;//60cyc
		nRotativeWorkPosition						: DINT	:= 450;	//80 grades
		bSetValues									: BOOL;
		bCycError									: BOOL;
		
		bCloseGuideGripper							: BOOL;
		bCloseFixtureGripper						: BOOL;
		
		nScaledLinearVel							: DINT;
		nScaledLinearAcc							: DINT;
		nScaledLinearSetPoint						: DINT;
		nScaledLinearTorque							: INT;
	
		nScaledRotativeVel							: DINT;
		nScaledRotativeAcc							: DINT;	
		nScaledRotativeSetPoint						: DINT;

		
///////////////////////////////////////CYCLE//////////////////////////////////////////////////	
		//INPUTS:
		bCycProcess									: BOOL;
		bAutoCycleAcknowledge						: BOOL;
		bAutoCycleRequest							: BOOL;
		bResetAutoCycle								: BOOL;
		bInitSecondPart								: BOOL;
		//OUTPUTS:
		bAutoCycleAcknowledgeRequest				: BOOL;
		bCycleProcessDone							: BOOL;
		bFirstPartDoneFlag							: BOOL;
		bOpenGuideGripper							: BOOL;
		
///////////////////////////////////////REPORT//////////////////////////////////////////////////	
		
		nDistanceSetPoint							: DINT;
		nDistanceTolerance							: DINT;
		bPass										: BOOL;
		bFail										: BOOL;
		MaxDistanceReached							: DINT;


END_STRUCT
END_TYPE

// ---- DUTs/04_SMAC/FUNCTIONS/ST_Phasing_Home.TcDUT
TYPE ST_Phasing_Home :
STRUCT
			//INPUTS:
		bEnable										: BOOL;
		bAcknowledge								: BOOL;
		bReset										: BOOL;	
		bFunctionRequest							: BOOL;

		//OUTPUTS:	
		bFunctionEnabled							: BOOL;
		bPhasingProcessDone							: BOOL;
		bHomingProcessDone							: BOOL;
		bAcknowledgeRequest							: BOOL;
		bHomeError									: BOOL;
		bPhasingError								: BOOL;
END_STRUCT
END_TYPE

// ---- DUTs/04_SMAC/I_O/ST_SMAC_I_O.TcDUT
TYPE ST_SMAC_I_O :
STRUCT

////////////////////////////////INPUTS///////////////////////////////////

inStatusWordLinear							AT %I*				: DINT; //CHECK TABLE IN MANUAL
inModeOfOperationLinear						AT %I*				: DINT;
inCurrentPositionLinear						AT %I*				: DINT;
inErrorIDLinear								AT %I*				: DINT;
inCurrentValueLinear						AT %I*				: INT;

inStatusWordRotative						AT %I*				: DINT; //CHECK TABLE IN MANUAL
inModeOfOperationRotative					AT %I*				: DINT;
inCurrentPositionRotative					AT %I*				: DINT;
inErrorIDRotative							AT %I*				: DINT;
inCurrentValueRotative						AT %I*				: INT;

inCurrentMacro								AT %I*				: INT;



////////////////////////////////OUTPUTS///////////////////////////////////

qnControlWordLinear							AT %Q*				: UINT; //CHECK TABLE IN MANUAL
qnModeOfOperationLinear						AT %Q*				: UINT; //CHECK TABLE IN MANUAL
qnSetPointLinear							AT %Q*				: DINT;
qnSetVelocityLinear							AT %Q*				: DINT;
qnSetAcceleraionLinear						AT %Q*      		: DINT;
qnSetMaxiumTorqueLinear						AT %Q*				: INT;

qnControlWordRotative						AT %Q*				: UINT; //CHECK TABLE IN MANUAL
qnModeOfOperationRotative					AT %Q*				: UINT; //CHECK TABLE IN MANUAL
qnSetPointRotative							AT %Q*				: DINT;
qnSetVelocityRotative						AT %Q*				: DINT;
qnSetAcceleraionRotative					AT %Q*      		: DINT;
qnSetMaxiumTorqueRotative					AT %Q*				: INT;

qnSetMacroNumber							AT %Q*				: INT;

////////////////////////////////////////////////////////////////////////////

sStatus					: ARRAY [0..20] OF STRING;
sModeOfOperation		: ARRAY [0..11] OF STRING;
sControlWord			: ARRAY [0..6] OF STRING; 	
 




END_STRUCT
END_TYPE

// ---- DUTs/04_SMAC/ST_Smac.TcDUT
TYPE ST_Smac :
STRUCT

	// Set Action
	bSet_PickScrew							:BOOL;											
	bSet_ScrewItIn							:BOOL;
	
	// Grippers CTRL
	bGripperA_Close							:BOOL;	// Channel 03 - Gripper A Close CMD		
	bGripperA_Open							:BOOL;	// Channel 04 - Gripper A Open CMD
	bGripperB_Close							:BOOL;	// Channel 05 - Gripper B Close CMD		
	bGripperB_Open							:BOOL;	// Channel 06 - Gripper B Open CMD

	// Grippers Feedback Sensors
	bGripperA_ClosedSensor					:BOOL;	// Channel 04 - Gripper A Closed Position Sensor
	bGripperB_ClosedSensor					:BOOL;	// Channel 05 - Gripper B Closed Position Sensor	
	


//--------------------------------------------------------------------------------------------------oldschoo1
	
END_STRUCT
END_TYPE

// ---- DUTs/05_ProcessCycle/E_ProcessCycle.TcDUT
{attribute 'qualified_only'}
{attribute 'strict'}
TYPE E_ProcessCycle :
(

	
IDLE					:=0,
AXIS_CMD_1				:=10,
WAIT_AXIS_CMD_1			:=15,
SMAC_CMD_1				:=20,
WAIT_SMAC_CMD_1			:=25,
AXIS_CMD_2				:=30,
WAIT_AXIS_CMD_2			:=35,
GRIPPERS_CMD_1			:=37,
WAIT_GRIPPERS_CMD_1		:=38,
CMD_SMAC_KISLR			:=40,
WAIT_SMAC_KISLR			:=45,
STORE_PROC_DATA			:=50,
Saving_DATA				:=53,
GRIPPERS_CMD_2			:=55,
WAIT_GRIPPERS_CMD_2		:=56,
CMD_KISLR				:=58,
WAIT_KISLR				:=59,
AXIS_CMD_3				:=60,
WAIT_AXIS_CMD_3			:=65,
AXIS_HOME				:=70,
WAIT_AXIS_HOME			:=75,
RESET_ALL_CMD			:=80

//----------------------------oldschoo1

);
END_TYPE

// ---- DUTs/05_ProcessCycle/ST_ProcessReport.TcDUT
TYPE ST_ProcessReport :
STRUCT
	

	// Time && Date
	sDate									:STRING;		// Record System Time&Date whenn proccess started
	sTime									:STRING;	
	
	// Kistler
	rKis_DistanceRecord						:REAL;   
	rKis_ForceRecord						:REAL;     
	rKis_HighestRecordedForce				:REAL;				// Maximum Force reached during the Press travel 
	rKis_LowestRecordedForce				:REAL;				// Maximum Force reached during the Press travel
	rKis_Settings_ForceUpperTreshold		:REAL;				// Setting value of the Upper Force Treshold for PASS/FAIL
	rKis_Settings_ForceLowerTreshold		:REAL;				// Setting value of the Lower Force Treshold for PASS/FAIL
	rKis_Settings_StartMeasurePoint			:REAL;				// Setting value of the Start Point of the Kistler travel
	rKis_Settings_ReservoirBottomPoint		:REAL;				// Setting value of the Bottom Point of the Kistler travel
	sKis_Result								:STRING;	
	bKis_Pass								:BOOL;				// TRUE if it was a PASS
	bKis_Fail								:BOOL;				// TRUE if it was a FAIL	
	
	
	// Smac 
	rSmac_MaxDistanceReached				:LREAL;
	rSmac_NumberOfCycles					:LREAL;
	rSmac_Settings_LinearVel				:LREAL;
	rSmac_Settings_LinearTorque				:LREAL;
	rSmac_Settings_RotativeVel				:LREAL;
	rSmac_Settings_LinearAcc				:LREAL;
	rSmac_Settings_RotativeAcc				:LREAL;
	sSmac_Result							:STRING;
	bSmac_Pass								:BOOL;					
	bSmac_Fail								:BOOL;	
	
	
	//-----------------------------------------------------------------------------------------------------------------------oldschoo1
	
	
END_STRUCT
END_TYPE

// ---- GVLs/ETHIP.TcGVL
{attribute 'qualified_only'}
VAR_GLOBAL
	Test6							AT %MB0				:DINT;
	Test7							AT %MB10			:DINT;
END_VAR

// ---- GVLs/GVL_CONSTANTS.TcGVL
VAR_GLOBAL CONSTANT
//SEBASTIAN ULLOA 22/07/25 INIT-----------------------------------------------------
//Colors HMI
	sWHITE                              :   STRING(40)  := '{"color":"rgba(255,255,255,255)"}';
    sBLACK                              :   STRING(40)  := '{"color":"rgba(0,0,0,1)"}';
    sYELLOW                             :   STRING(40)  := '{"color":"rgba(255,255,0,1)"}';
    sGREEN                             	:   STRING(40)  := '{"color":"rgba(70,166,63,1)"}';
	sLGREEN                             :   STRING(40)  := '{"color":"rgba(58,211,20,1)"}';
    sORANGE                             :   STRING(40)  := '{"color":"rgba(255,153,51,1)"}';
    sNYPROORANGE                        :   STRING(40)  := '{"color":"rgba(255,140,0,1)"}';
    sRED                                :   STRING(40)  := '{"color":"rgba(255,0,0,1)"}';
	sLRED                               :   STRING(40)  := '{"color":"rgba(233,53,44,1)"}';
    sBLUE                               :   STRING(40)  := '{"color":"rgba(0,0,255,1)"}';
	sLBLUE                              :   STRING(40)  := '{"color":"rgba(0,162,232,1)"}';
    sGREY                               :   STRING(40)  := '{"color":"rgba(164,158,158,1)"}';
    sScreenGREY                         :   STRING(40)  := '{"color":"rgba(225,225,225,1)"}';
    sDARKGREY                           :   STRING(40)  := '{"color":"rgba(50,50,50,1)"}';
    sPURPLE                             :   STRING(40)  := '{"color":"rgba(128,0,128,1)"}';
    sVIOLET                             :   STRING(40)  := '{"color":"rgba(204,153,255,1)"}';
    sTRANSP                             :   STRING(40)  := '{"color":"rgba(255,255,255,0)"}';
    sGREENPass                          :   STRING(40)  := '{"color":"rgba(0,153,51,1)"}';
    sREDFail                            :   STRING(40)  := '{"color":"rgba(244,68,68,255)"}';
    sBLUEInProgress                     :   STRING(40)  := '{"color":"rgba(54,100,221,1)"}';
	sGREENISHTEAColor					:	STRING(40)  := '{"color":"rgba(60,192,134,255)"}'	;

	nBLACK								: 	DWORD 	:= 	16#FF000000;	 // format: TTRRGGBB where T -> 00 = full transparency and FF = full opaque
	nWHITE								: 	DWORD 	:= 	16#FFFFFFFF;
	nYELLOW								: 	DWORD 	:= 	16#FFFFFF00; 
	nGREEN								: 	DWORD 	:= 	16#FF008A00;
	nLIGHTGREEN                         :   DWORD   :=  16#FF98FB89;
	nORANGE								: 	DWORD 	:= 	16#FFFFA500;
	nNYPROORANGE						:	DWORD	:=	16#FFF05322;
	nRED								: 	DWORD 	:= 	16#FFFF0000;
	nBLUE								: 	DWORD 	:= 	16#FF0000FF;
	nLIGHTBLUE                          :   DWORD   :=  16#FF08ADF4;
	nGREY								: 	DWORD 	:= 	16#FFA9A9A9;	
	nDARKGREY							:	DWORD	:=	16#FF808080;
	nPURPLE								:	DWORD	:=	16#FF800080;
	nVIOLET								:	DWORD	:=	16#FFEE82EE;
	nTRANSP								:	DWORD	:=	16#00FFFFFF;	// full transparent WHITE
	
	nLCColNormal						:	DWORD	:= 16#10008A00;		// light curtain green
	nLCColBroken						:	DWORD	:= 16#64FF0000;		// light curtain red	
//SEBASTIAN ULLOA 22/07/25 END-----------------------------------------------------
END_VAR

// ---- GVLs/GVL_MODULES.TcGVL
VAR_GLOBAL
	

	// Y-Axis
	stY_Axis			:ST_Y_Axis;
	
	CMD_Axis			:ST_ModuleCMD;
	Axis_STATUS			:ST_ModuleStatus;
	
	// Kistler
	stKistler			:ST_Kistler;

	CMD_Kistler			:ST_ModuleCMD;
	Kistler_STATUS		:ST_ModuleStatus;
	
	// Smac
	stSmacIO			: ST_SMAC_I_O; //It suppose to be in GVL_IO
	stSmac				: ST_Smac;
	
	CMD_Smac			:ST_ModuleCMD;
	Smac_STATUS			:ST_ModuleStatus;	
	
	
//--------------------------------------------oldschoo1	
	
END_VAR

// ---- GVLs/GVL_PERSISTENT.TcGVL
{attribute 'qualified_only'}
VAR_GLOBAL PERSISTENT


	// Y-Axis Parameters
										//Position Offsets must be in small increments, never bigger then 1.3mm
	fPositions_Offset					:ARRAY [1..3]OF LREAL;//HMI offset for only: [1]-Picking Screw,[2]-Press && Screwing Actions
	
	
	// Kistler Parameters - For Force evaluation PLC logic	 (only Bottom Position will be send to the controller)
	rKistlerForce_UpperLimit			:REAL;//:= 75.0;	//HMI parameter - Force Upper threshold limit for PASS/FAIL
	rKistlerForce_LowerLimit			:REAL;//:=  7.0;	//HMI parameter - Force Lower threshold limit for PASS/FAIL
	rKistlerForce_Speed					:REAL;//:=	9.3 mm/s;	//HMI parameter - Position where Press Cylinder starts touching Reservoir

	
	rMeasurementTolerance				:REAL;//:=  3.0;	//HMI parameter - Force Measurement Tolerance
	rReservoir_ContactPosition			:REAL;//:=	 5.2;	//HMI parameter - Position where Press Cylinder starts touching Reservoir
	rReservoir_BottomPosition			:REAL;//:=	28.6;	//HMI parameter - Position where the pressure cylinder touches the end of Reservoir.
	rReservoir_Bottomlimitoffset		:REAL;//:=	0.5;	//HMI parameter - Offset to validate the force up to the position where the pressure cylinder finishes touching the Reservoir
	DatosHistory 						:ARRAY [1..100,1..100] OF Stpoint;  // Output array with captured data
	GraphDataHistorystorage				:ARRAY [1..100,1..100] OF Stpoint;
	// Kistler Parameters
	
	
	
	// Proccess Counter
	stProccessReportLog					:ARRAY [1..250]OF ST_ProcessReport;
	
	
	
	//HMI
	stUserLogHMI				: ARRAY[0..250] OF ST_UserLogHMI;
	UserId						: UINT;
	bSMACEnable					: BOOL;
	
	//Statistics
	nSmacGoodParts				: DINT;
	nKistlerGoodParts			: DINT;
	nSmacTotalGoodParts			: DINT;
	nKistlerTotalGoodParts		: DINT;
	nSmacBadParts				: DINT;
	nKistlerBadParts			: DINT;
	nSmacTotalBadParts			: DINT;
	nKistlerTotalBadParts		: DINT;
	
	nSmacRotativeSetPoint		: DINT;
	
	//-----------------------------------------------------------------------------------------------------------------------oldschoo1
	h							: INT:=1;
END_VAR

// ---- GVLs/GVL_HMI.TcGVL
{attribute 'qualified_only'}
VAR_GLOBAL
	
	(*-----------------------------------------------------------------------------------------------------------------*)
	// HMI System Info
	sSoftwareVersion					: STRING;
	sSoftwareDate						: STRING := 'Jul 2025' ;
	sTC3Version							: STRING := 'v3.1.4024.53, Runtime v3.1.4024.53' ;
	sVisualStudioVersion				: STRING := 'TcXaeShell' ;
	sSystemName							: STRING := 'Stopper Insertion And Screw Station' ;
	sProjectID							: STRING := 'TE1096-04-SISS' ;
	sHMIServer                			: STRING := '' ;
	//sIPAddress						: STRING;// := '192.168.7.170'; (Should NOT available on HMI) -o1
	ntAMSNetID							: T_AmsNetId :='172.18.233.151.1.1';
	sSafetyCRC							: STRING;
	sTrayNameAndTotalTrays				: STRING;
	sMessageToOperator					: STRING;
	
	(*-----------------------------------------------------------------------------------------------------------------*)
	
	
	(*-----------------------------------------------------------------------------------------------------------------*)
	
	
	
	
	(*-----------------------------------------------------------------------------------------------------------------*)
	// Settings Menu for the Modules
	
	// Y-Axis
	//MANUAL
	bMoveToPos							:BOOL;
	bY_AxisPosition1					:BOOL;
	bY_AxisPosition2					:BOOL;
	bY_AxisPosition3					:BOOL;
	bY_HomePosition						:BOOL;
	bEnableManualMode					:BOOL;
	rtrigManualMode						:R_TRIG;
	rTrigManualModeOff					:ARRAY[0..4] OF R_TRIG;
	nRegionMain							:DINT;
	nRegionSetting						:DINT;
	bManualModeOff						:ARRAY[0..4] OF BOOL;
	bY_AxisInPosition1					:BOOL;
	bY_AxisInPosition2					:BOOL;
	bY_AxisInPosition3					:BOOL;
	bY_AxisInHomePosition				:BOOL;
	bY_AxisInPosition1Man				:BOOL;
	bY_AxisInPosition2Man				:BOOL;
	bY_AxisInPosition3Man				:BOOL;
	bY_AxisInHomePositionMan			:BOOL;
	GraphData							:ARRAY [1..1,1..100] OF Stpoint;
	GraphDataHistory					:ARRAY [1..1,1..100] OF Stpoint;
	
	
	// Kistler
	rKistlerLiveReading_X				:REAL;	//Travel
	rKistlerLiveReading_Y				:REAL;	//Force
	bKistlerCycle						:BOOL;
	rKistlerAnimationMan				:LREAL;
	rKistlerAnimationCyc				:LREAL;
	rKisterldistanceHMI					:REAL; 
	rKisterlForceHMI					:REAL; 
	
	
	// Smac
	nCurrentDistanceSmac				:LREAL;
	nCurrentVelocity					:LREAL;
	rSmacAnimationMan					:LREAL;
	rSmacAnimationCyc					:LREAL;
	
	rScrewAnimation						:LREAL;
	bScrewAnimation						:BOOL;
	bScrewPartPresent					:BOOL;
	bSmacCyc1							: BOOL;
	bSmacCyc2							: BOOL;
	bSmacHOME							: BOOL;
	bSmacSetValue						: BOOL;
	
	bLinearServoEnabled					: BOOL;
	bLinearHomingSuccess				: BOOL;
	bLinearPhasingSuccess				: BOOL;
	bLinearError						: BOOL;
	
	bRotativeServoEnabled				: BOOL;
	bRotativeHomingSuccess				: BOOL;
	bRotativePhasingSuccess				: BOOL;
	bRotativeError						: BOOL;
	
	bSmacSTO1Fault						: BOOL;
	bSmacSTO2Fault						: BOOL;
	bSmacGeneralFault					: BOOL;
	bSmacOverCurrentFault				: BOOL;
	
	(*-----------------------------------------------------------------------------------------------------------------*)
	//General
	aManualScreens						: ARRAY[0..1] OF STRING(200);
	aSettingScreens						: ARRAY[0..2] OF STRING(200);
	aIOScreens							: ARRAY[0..16] OF STRING(200);
	bResetSmacGoodParts					: BOOL;
	bResetKistlerGoodParts				: BOOL;
	bResetSmacBadParts					: BOOL;
	bResetKistlerBadParts				: BOOL;
	
	//User Log, Shut down, Quit HMI
	bQuitHmi						: BOOL;
	bKistlerHMI						: BOOL;
	sUserGroup						: STRING;
	sUserGroup2						: STRING;
	sUserName						: STRING;
	bLogOut							: BOOL;
	bUserLogedIntSignal				: BOOL;
	bShutDown						: BOOL; 
	//Alarns
	aEventTexts							: ARRAY [0..767] OF T_MaxSTring; //Event texts - set only once
	bEventTextsSet						: BOOL;
	aEventFlags							: ARRAY [0..767] OF BOOL;		//All event states combined from master na stations
	aActiveEvents						: ARRAY [0..39] OF T_MaxSTring;	//Active events - connected to Alarm scree in HMI	
	stActiveEventsHMI					: ARRAY [0..39] OF ST_ActiveEventsHMI;
	


END_VAR
VAR_GLOBAL PERSISTENT
	stAlarmHistory				:ARRAY [00..250] OF ST_AlarmHistory;
	aEventLog					:ARRAY [0..250] OF T_MaxSTring;	//Event log - connected to alarm history in HMI	
	aTimeLog					:ARRAY [0..250] OF T_MaxSTring;
	aDateLog					:ARRAY [0..250] OF T_MaxSTring;
	sSystemDate					: STRING;
	sSystemTime					: STRING;
	
END_VAR

// ---- GVLs/GVL_IO.TcGVL
{attribute 'qualified_only'}
VAR_GLOBAL

	fbTerminalInfo												:ARRAY[0..20] OF FB_TerminalInfo;
	//-----------------------------------------------------------------------------------------------------------------------oldschoo1
   	// TERMINAL 1 _ EK1100 - EtherCAT Coupler

	nEK1100State							AT %I*				:UINT;	// Terminal INFO Data	
	sEK1100Status												:STRING(200);
	
	//-------------------------------------------------------------------------------------------------------------------------License
	// TERMINAL 2 _ EL6070-0033	- License Key Terminal for TC3
	
	nEL6070State							AT %I*				:UINT;	// Terminal INFO Data	
	sEL6070Status												:STRING(200);

	
(**************************************************** Safety - I/O *****************************************************************)	
	//-------------------------------------------------------------------------------------------------------------------------SAFETY
	// TERMINAL 3 _ EL6910 - Safety PLC - Virtual Channels
	
		//Q
	qsSafetyRun                          	AT %Q*          	:BOOL;  // VirtualCh - Start Safety CMD
	qsSafetyErrorAck						AT %Q* 				:BOOL;	// VirtualCh - Safety Error Acknowledge

	qsTwoHandsMonitoring                    AT %Q*          	:BOOL;  // VirtualCh - 2Hands needed to trigger Proccessing 
	qsLightBeam_MutingActive				AT %Q*				:BOOL;	// VirtualCh - SICK Safety LightBeam - Muting active
	qsLockDoorCMD							AT %Q*				:BOOL;	// VirtualCh - CMD to lock the Door
	
	
		//I
	isSafetyRunning                         AT %I*          	:BOOL;  // VirtualCh - TwinSAFE running
	isSafetyFB_Error	 					AT %I*				:BOOL;	// VirtualCh - TwinSAFE modules Feedback Error
	isSafetyCom_Error 						AT %I*	 			:BOOL;	// VirtualCh - TwinSAFE Communication error	
	isSafety_OK								AT %I*				:BOOL;	// VirtualCh - All safety gear OK
    isEStop_OK	                         	AT %I*          	:BOOL;  // VirtualCh - E-Stop OK
	isDoorClosed							AT %I*				:BOOL;	// VirtualCh - Door Closed
	isDoorLocked							AT %I*				:BOOL;	// VirtualCh - Door Locked
	isLightBeam_NotCrossed					AT %I*				:BOOL;	// VirtualCh - SICK Safety LightBeam - Not crosed
	isLightBeam_OK							AT %I*				:BOOL;	// VirtualCh - SICK Safety LightBeam - Muted
	isTwoHands_SIGNAL						AT %I*				:BOOL;	// VirtualCh - TwoHands - Both Buttons activated

		//Status*
	nEL6910State							AT %I*				:UINT;	// Terminal INFO Data	
	sEL6910Status												:STRING(200);

	
	//---IN--------------------------------------------------------------------------------------------------------------------------I
	// TERMINAL 4 _ EL1918 - 8 Channel Digital Safety Inputs
	
	iE_Stop_Ch1								AT %I*				:BOOL;	// Channel 1 - E-Stop ch1
	iE_Stop_Ch2								AT %I*				:BOOL;	// Channel 2 - E-Stop ch2                               	
	iResetButton							AT %I*				:BOOL;	// Channel 3 - Reset Button	
	iDoorInterlock_Ch1						AT %I*				:BOOL;	// Channel 4 - Door Closed ch1
	iDoorInterlock_Ch2						AT %I*				:BOOL;	// Channel 5 - Door Closed ch2	                                	
	iDoorInterlock_FB						AT %I*				:BOOL;	// Channel 6 - Door Feedback Sig.
	iIndraDrive_Contactor_FB				AT %I*				:BOOL;	// Channel 7 - Kistler drive Safety Contactor Feedback
	iSmacSTO_FB								AT %I*				:BOOL;	// Channel 8 - SMACK Safe Torque OFF Feedback
	
		//Status*
	nEL1918_1State							AT %I*				:UINT;	// Terminal INFO Data	
	sEL1918Status												:STRING(200);
	
	
	//---IN--------------------------------------------------------------------------------------------------------------------------I
	// TERMINAL 5 _ EL1918 - 8 Channel Digital Safety Inputs
	
	iTouchBtn_1_NC							AT %I*				:BOOL;	// Channel 1 - Safety Touch Button 1 
	iTouchBtn_2_NC							AT %I*				:BOOL;	// Channel 2 - Safety Touch Button 2                               	
	iTouchBtn_1_NO							AT %I*				:BOOL;	// Channel 3 - Safety Touch Button 1
	iTouchBtn_2_NO							AT %I*				:BOOL;	// Channel 4 - Safety Touch Button 2
	iPilz2_FB								AT %I*				:BOOL;	// Channel 5 - Pilz Safety Relay 2 Feedback
	iAxis_1_SafetyRelayFB					AT %I*				:BOOL;	// Channel 6 - AXIS 1 Safety Relay Feedback
	iSafetyBeam_Signal						AT %I*				:BOOL;	// Channel 7 - SICK Safety LightBeam Signal
																		// Channel 8 - Spare

		//Status*                      	
	nEL1918_2State							AT %I*				:UINT;	// Terminal INFO Data	
	sEL1918_2Status												:STRING(200);
	
	
	//---OUT-------------------------------------------------------------------------------------------------------------------------Q
	// TERMINAL 6 _ ELEL2904 - 4 Channel Digital Safety Outputs
	
	qPilz1_Coil								AT %Q*				:BOOL;	// Channel 1 - PSR1 Pilz Coil                                	
	qIndraDrive_EStop						AT %Q*				:BOOL;	// Channel 2 - Kistler drive Safety Contactor E-Stop Sig.
	qPilz2_EStop							AT %Q*				:BOOL;	// Channel 3 - PSR2 Pilz E-Stop Sig.
	qDoorInterlock_CMD						AT %Q*				:BOOL;	// Channel 4 - Door Lock Solenoid
	
		//Status*
	nEL2904_1State							AT %I*				:UINT;	// Terminal INFO Data	
	sEL2904_1Status												:STRING(200);
	
	
	//---OUT-------------------------------------------------------------------------------------------------------------------------Q
	// TERMINAL 7 _ ELEL2904 - 4 Channel Digital Safety Outputs
	
	qSmacSTO_Ch1							AT %Q* 				:BOOL;	// Channel 1 - SMAC SafeTorque OFF - Input 1
	qSmacSTO_Ch2							AT %Q* 				:BOOL;	// Channel 2 - SMAC SafeTorque OFF - Input 2	                                	
																		// Channel 3 - Spare
	qAxis_1_SafetyRelayCoil					AT %Q* 				:BOOL;	// Channel 4 - AXIS 1 Safety Relay Coil

		//Status* 
	nEL2904_2State							AT %I*				:UINT;	// Terminal INFO Data	
	sEL2904_2Status												:STRING(200);

	
	
	
(**************************************************** PLC - I/O *********************************************************************)
										
	//---IN-------------------------------------------------------------------------------------------------------------------PLC I/O
	// TERMINAL 8 _ EL1809 - 16 Channel Digital Input Terminal
	
	iStartButton							AT %I*				:BOOL;	// Channel 01 - Start Button 
	iStopButton   	 						AT %I*				:BOOL;	// Channel 02 - Stop Button
	iPSU_1_OK								AT %I*	 			:BOOL;	// Channel 03 - Power Supply Unit 1 OK
	iPSU_2_OK								AT %I*	 			:BOOL;	// Channel 04 - Power Supply Unit 2 OK
	iPSU_3_OK								AT %I*	 			:BOOL;	// Channel 05 - Power Supply Unit 3 OK
																		// Channel 06 - Spare
																		// Channel 07 - Spare
																		// Channel 08 - Spare
	iKistlerCTRL_FB1						AT %I*	 			:BOOL;	// Channel 09 - Kistler CTRL - Feedback Signal 1	
	iKistlerCTRL_FB2						AT %I*	 			:BOOL;	// Channel 10 - Kistler CTRL - Feedback Signal 2	
	iKistlerCTRL_FB3						AT %I*	 			:BOOL;	// Channel 11 - Kistler CTRL - Feedback Signal 3	
																		// Channel 12 - Spare   
	iSmacCTRL_FB1							AT %I*	 			:BOOL;	// Channel 13 - SMAC CTRL - Feedback Signal 1	
	iSmacCTRL_FB2							AT %I*	 			:BOOL;	// Channel 14 - SMAC CTRL - Feedback Signal 2	
	iSmacCTRL_FB3							AT %I*	 			:BOOL;	// Channel 15 - SMAC CTRL - Feedback Signal 3
																		// Channel 16 - Spare 

		//Status*	
	nEL1809_1State							AT %I*				:UINT;	// Terminal INFO Data	
	sEL1809_1Status												:STRING(200);
	

	//---IN--------------------------------------------------------------------------------------------------------------------------I
	// TERMINAL 9 _ EL1809 - 16 Channel Digital Input Terminal
	
	iPuck_PresentSensor						AT %I*				:BOOL;	// Channel 01 - Puck Fixture present Sensor
	iPartA_PresentSensor   	 				AT %I*				:BOOL;	// Channel 02 - Part A present inside Fixture
	iPartB_PresentSensor   	 				AT %I*				:BOOL;	// Channel 03 - Part B present inside Fixture
	iGripperA_ClosedSensor					AT %I*	 			:BOOL;	// Channel 04 - Gripper A Closed Position Sensor
	iGripperB_ClosedSensor					AT %I*	 			:BOOL;	// Channel 05 - Gripper B Closed Position Sensor
	iPartC_PresentSensor   	 				AT %I*				:BOOL;	// Channel 06 - Part C present inside Fixture
																		// Channel 07 - Spare
																		// Channel 08 - Spare
																		// Channel 09 - Spare
																		// Channel 10 - Spare
																		// Channel 11 - Spare
																		// Channel 12 - Spare
																		// Channel 13 - Spare
																		// Channel 14 - Spare
																		// Channel 15 - Spare
																		// Channel 16 - Spare

		//Status*	
	nEL1809_2State							AT %I*				:UINT;	// Terminal INFO Data
	sEL1809_2Status												:STRING(200);
	
	
	//---OUT-------------------------------------------------------------------------------------------------------------------------Q
	// TERMINAL 10 _ EL2809	- 16 Channel Digital Output Terminal
	
	qStartButton_LED						AT %Q*				:BOOL;	// Channel 01 - Start Button Indicator LED
	qResetButton_LED						AT %Q* 				:BOOL;	// Channel 02 - Stop Button Indicator LED
	qGripperA_Close							AT %Q*	 			:BOOL;	// Channel 03 - Gripper A Close CMD		
	qGripperA_Open							AT %Q*	 			:BOOL;	// Channel 04 - Gripper A Open CMD
	qGripperB_Close							AT %Q*	 			:BOOL;	// Channel 05 - Gripper B Close CMD		
	qGripperB_Open							AT %Q*	 			:BOOL;	// Channel 06 - Gripper B Open CMD
	qCycleIndicator_RedLED					AT %Q*	 			:BOOL;	// Channel 07 - Cycle Indicator LED - Red
	qCycleIndicator_GreenLED				AT %Q*	 			:BOOL;	// Channel 08 - Cycle Indicator LED - Green
	qKistlerCTRL_Sig1						AT %Q*	 			:BOOL;	// Channel 09 - Kistler CTRL Signal 1
	qKistlerCTRL_Sig2						AT %Q*	 			:BOOL;	// Channel 10 - Kistler CTRL Signal 2
	qKistlerCTRL_Sig3						AT %Q*	 			:BOOL;	// Channel 11 - Kistler CTRL Signal 3
	qKistlerCTRL_Sig4						AT %Q*	 			:BOOL;	// Channel 12 - Kistler CTRL Signal 4	
	qSmacCTRL_Sig1							AT %Q*	 			:BOOL;	// Channel 13 - Smac CTRL Signal 1	
	qSmacCTRL_Sig2							AT %Q*	 			:BOOL;	// Channel 14 - Smac CTRL Signal 2
	qSmacCTRL_Sig3							AT %Q*	 			:BOOL;	// Channel 15 - Smac CTRL Signal 3
																		// Channel 16 - Spare
		//Status*
	nEL2809State							AT %I*				:UINT;	// Terminal INFO Data
	sEL2809Status												:STRING(200);


(***************************************************************************************************************************************)
	
	//---------------------------------------------------------------------------------------------------------------------------DRIVE
	// TERMINAL 11 _ EL9576 - Brake Chopper Terminal

		//Status*
	nEL9576State							AT %I*				:UINT;	// Terminal INFO Data
	sEL9576Status												:STRING(200);
	
	//---------------------------------------------------------------------------------------------------------------------------DRIVE
	// TERMINAL 12 _ EL7211-0010 - Servo Motor Drive
	
		//Status*
	nEL7211State							AT %I*				:UINT;	// Terminal INFO Data
	sEL7211Status												:STRING(200);	

	
(**************************************************** EtherCAT **********************************************************************)
	
	//-------------------------------------------------------------------------------------------------------------------------KISTLER
	// BOX 13 _ maXYnos - Drive and Force Sensor for Kistler Press
	
	iStatusBytes                           AT %I*          		:ARRAY [0..199] OF BYTE;	//Status
	qControlBytes                          AT %Q*          		:ARRAY [0..199] OF BYTE;	//CMDs
	
		//Status*
	nKistlermaXYmosState				   AT %I*		   		:UINT;	// Terminal INFO Data
	sKistlermaXYmosStatus								   		:STRING(200);	

	//----------------------------------------------------------------------------------------------------------------------------SMAC
	// BOX 14 _ SMAC - Linear amd Rotative axis for screw part
	
	
	//------------------------------------------------------------------------------------------------------------------------------128

	
END_VAR

// ---- GVLs/GVL_MASTER.TcGVL
VAR_GLOBAL

	// PowerUP 
	tonSystemPowerUP							:Tc2_Standard.TON;
	tSystemPowerUP_Time							:TIME:=T#35S;
	bSystemPoweringUP							:BOOL:=TRUE; //Global System PowerUP Flag
	
	bFirstRun									:BOOL:=TRUE;
	tonFirstRun									: TON;
	
	sSystemDate									:STRING;
	sSystemTime									:STRING;
	
	// Master m/c Status
	stMachineStatus								:ST_MachineStatus;
	stSafety									:ST_SafetyPLC;
	stMasterCTRL								:ST_MasterCTRL;
	
	
	//---------------------------------------------------------------------------------------------*
											//I:
	// CTRL Buttons: 
	bStartButtonRisingEdge				        :BOOL;	// Start button
	bStartButtonFallingEdge				        :BOOL;
	bStopButtonRisingEdge						:BOOL;	// Stop button
	bStopButtonFallingEdge						:BOOL;
	bResetButtonRisingEdge						:BOOL;	// Reset button
	bResetButtonFallingEdge						:BOOL;

	// Master Input Sensors
	bPuck_Present								:BOOL;	// Puck Fixture present - Sensor
	bGearBox_Present   	 						:BOOL;	// GearBox present inside Fixture
	bScrew_Present   	 						:BOOL;	// Screw present inside Fixture
	bReservoir_Present   	 					:BOOL;	// Reservoar present inside Fixture

											//Q:
	//Cycle Indicator LED
	bCycleIndicator_Green						:BOOL;	// Processing in progress
	bCycleIndicator_Red							:BOOL;	// Processing compleeted
	
	bOpenGrippers								: BOOL;
	
	
	//--------------------------------Alarms--------------------------------------------------------*
	
	stAlarms                        			: ARRAY [0..3] OF ST_Events;

	//--------------------------------------------------------------------------------------oldschoo1
	
END_VAR

// ---- GVLs/GVL_UTILITIES.TcGVL
VAR_GLOBAL
	
	// System Oscilator Pulses at 2ms tick
	
	// 50% Duty Cycle
	bFlash05Hz						:BOOL;
	bFlash1Hz						:BOOL;
	bFlash2Hz						:BOOL;
	bFlash5Hz				   		:BOOL;
	bFlash10Hz						:BOOL;
	bFlash50Hz        		  		:BOOL;
	bFlash250Hz      	      		:BOOL;

	//Frictions
	bFlash1p52Hz					:BOOL;	//1.52Hz
	bFlash1p85Hz					:BOOL;	//1.85Hz
	bFlash1p33Hz					:BOOL;	//1.33Hz
	bFlash1p2Hz						:BOOL;	//1.19Hz
	
	// 70/30 Duty Cycle
	bFlash1Hz_7030					:BOOL;

	// 80/20 Duty Cycle
	bFlash1Hz_8020					:BOOL;
	
//--------------------------------------------oldschoo1	
	
END_VAR

// ---- POUs/MAIN.TcPOU
PROGRAM MAIN
VAR
	// 
	

	//----------------------------------------------------------------------oldschoo1
END_VAR

(* 	for Jabil, Bray @ Tegan Innovations, Waterford - July2025. Ireland
 	m/c TE1096-04 SISS _rev1.0
	>> design by oldschoo1
	>> smac and hmi by seb	*)

 
// Calling:
A_Master();
   A_HMI();
D_FaultHandling(); 
   
//Get System Time
//PRG_SysTime();
PRG_MasterSystemTime();
//--------------------------------------------------------------------------oldschoo1

END_PROGRAM

// ---- POUs/00_MASTER/A_Master.TcPOU
PROGRAM A_Master
VAR

	// Buttons One-Shot Triggers:
	rtrigStartButton					:Tc2_Standard.R_TRIG;
	ftrigStartButton					:Tc2_Standard.F_TRIG;
	rtrigResetButton					:Tc2_Standard.R_TRIG;
	ftrigResetButton					:Tc2_Standard.F_TRIG;	
	rtrigStopButton					    :Tc2_Standard.R_TRIG;
	ftrigStopButton					    :Tc2_Standard.F_TRIG;

	
	//Write Persistent Data 
	fbWritePersistent					:Tc2_Utilities.FB_WritePersistentData;
	tonWritePeristentTrig				:Tc2_Standard.TON;
	bWritePersistentTrigger				:BOOL;	
	bWritePersistentError				:BOOL;
	bWritePersistentBusy				:BOOL;
	bWritePersistentErrID				:UDINT;
	tWritePersistentPeriod				:TIME := T#1M;	
	
	//----------------------------------------------------------------oldschoo1
	fbEventLogger						:	FB_EventLog;
	i                       :INT; //Int to handle user log index	
	k						:INT; //Int to handle user log index
	j						:INT;
	l						:INT;
	
END_VAR

// System PowerUP CTRL
tonSystemPowerUP(IN:=bSystemPoweringUP, PT:=tSystemPowerUP_Time);
IF tonSystemPowerUP.Q THEN 
bSystemPoweringUP:=FALSE;
 END_IF

tonFirstRun( IN := bFirstRun, PT := T#1S);

//
// Call Module's Actions:
			a_Map_Inputs();
	   b_Map_CtrlButtons();
	   
		  d_Call_Modules();
		  
		   f_Map_Outputs();
	   g_Map_StatusLamps();
  h_Write_PersistentData();
 			j_ManualMode();
  
//-------------------------oldschoo1

fbEventLogger(	bEnable       	:= PRG_MasterSystemTime.bReadyToRead AND NOT bSystemPoweringUP,
			    sDateTime     	:= PRG_MasterSystemTime.sDateTimeSpaces,
			    aEventFlags   	:= GVL_HMI.aEventFlags,
			    aEventTexts   	:= GVL_HMI.aEventTexts,
			    aActiveEvents 	:= GVL_HMI.aActiveEvents,
			    aEventLog     	:= GVL_HMI.aEventLog,
				siDate			:= GVL_MASTER.sSystemDate,
				siTime			:= GVL_MASTER.sSystemTime,
				soDate			:= GVL_HMI.aDateLog,
				soTime			:= GVL_HMI.aTimeLog
);

IF GVL_UTILITIES.bFlash250Hz THEN
FOR j := 0 TO 39 DO
	
GVL_HMI.stActiveEventsHMI[j].sActiveEvents := GVL_HMI.aActiveEvents[j];
END_FOR
FOR l:=0 TO 250 DO
	
	GVL_HMI.stAlarmHistory[l].sEventlog 	:= GVL_HMI.aEventLog[l];
	GVL_HMI.stAlarmHistory[l].sDate		:= GVL_HMI.aDateLog[l];
	GVL_HMI.stAlarmHistory[l].sTime		:= GVL_HMI.aTimeLog[l];
END_FOR
ELSE 
	
j:=0; 
l:=0;
END_IF

ACTION a_Map_Inputs:
// Safety Inputs
GVL_MASTER.stSafety.bSafety_OK						:= GVL_IO.isSafety_OK;
GVL_MASTER.stSafety.bDoorClosed						:= GVL_IO.isDoorClosed;
GVL_MASTER.stSafety.bDoorLocked						:= GVL_IO.isDoorLocked;
GVL_MASTER.stSafety.bEStop_OK						:= GVL_IO.isEStop_OK;
GVL_MASTER.stSafety.bLightBeam_Crossed				:= NOT GVL_IO.isLightBeam_NotCrossed;
GVL_MASTER.stSafety.bTwoHands_Signal				:= GVL_IO.isTwoHands_SIGNAL;



// Master Machine CTRL Inputs
GVL_MASTER.bPuck_Present							:= GVL_IO.iPuck_PresentSensor;
GVL_MASTER.bReservoir_Present						:= GVL_IO.iPartA_PresentSensor;
GVL_MASTER.bScrew_Present							:= GVL_IO.iPartB_PresentSensor;
GVL_MASTER.bGearBox_Present							:= GVL_IO.iPartC_PresentSensor;



// Y-Axis Inputs
GVL_MODULES.stY_Axis.bAxis_1_SafetyRelayFB			:= GVL_IO.iAxis_1_SafetyRelayFB;



// Kistler Inputs
GVL_MODULES.stKistler.st_TelegramDataIn				:= GVL_IO.iStatusBytes;
GVL_MODULES.stKistler.bKistlerCTRL_FB1				:= GVL_IO.iKistlerCTRL_FB1;						
GVL_MODULES.stKistler.bKistlerCTRL_FB2				:= GVL_IO.iKistlerCTRL_FB2;						 
GVL_MODULES.stKistler.bKistlerCTRL_FB3				:= GVL_IO.iKistlerCTRL_FB3;							



// Smac Inputs
GVL_MODULES.stSmac.bGripperA_ClosedSensor			:= GVL_IO.iGripperA_ClosedSensor;
GVL_MODULES.stSmac.bGripperB_ClosedSensor			:= GVL_IO.iGripperB_ClosedSensor;


//----------------------------------------------------------------------------------oldschoo1
END_ACTION

ACTION b_Map_CtrlButtons:

//Start button
rtrigStartButton(CLK:= GVL_IO.iStartButton,	Q=>bStartButtonRisingEdge);
ftrigStartButton(CLK:= GVL_IO.iStartButton,	Q=>bStartButtonFallingEdge);

// Stop button
rtrigStopButton(CLK:= NOT GVL_IO.iStopButton,  Q=>bStopButtonRisingEdge);
ftrigStopButton(CLK:= NOT GVL_IO.iStopButton,  Q=>bStopButtonFallingEdge);

// Reset button
rtrigResetButton(CLK:= GVL_IO.iResetButton, 	Q=>bResetButtonRisingEdge);
ftrigResetButton(CLK:= GVL_IO.iResetButton, 	Q=>bResetButtonFallingEdge);


//-------------------------------------------------------------------oldschoo1
END_ACTION

ACTION c_Read_Statuses:
//Handshake In
Y_Master_Y_Axis(STATUS => GVL_MODULES.Axis_STATUS);
K_Master_Kistler(STATUS => GVL_MODULES.Kistler_STATUS);
S_Master_SMAC(STATUS => GVL_MODULES.Smac_STATUS);
//--------------------------------------------oldschoo1
END_ACTION

ACTION d_Call_Modules:
// Call Modules Masters: ----------------------------------------*

			B_Safety();				// Safety PLC Module
							
	 c_Read_Statuses();
	  C_Machine_Ctrl();				// Master Module MachineCTRL
	 	e_Write_Cmds();
					
	 Y_Master_Y_Axis();				// Module for Y-Axis
   	   S_Master_SMAC();				// Module for Smac
	K_Master_Kistler();				// Module for Kistler	
   
//-------------------------------------------------------oldschoo1
END_ACTION

ACTION e_Write_Cmds:
//Handshake Out
Y_Master_Y_Axis(CMD := GVL_MODULES.CMD_Axis);
K_Master_Kistler(CMD := GVL_MODULES.CMD_Kistler);
S_Master_SMAC(CMD := GVL_MODULES.CMD_Smac);
//-----------------------------------------oldschoo1
END_ACTION

ACTION f_Map_Outputs:

// Safety Outputs
GVL_IO.qsSafetyRun								:= GVL_MASTER.stSafety.bRunSafety;
GVL_IO.qsSafetyErrorAck							:= GVL_MASTER.stSafety.bAckSafetyError;
GVL_IO.qsLockDoorCMD 							:= GVL_MASTER.stSafety.bLockDoor_CMD;
GVL_IO.qsLightBeam_MutingActive					:= GVL_MASTER.stSafety.bLightBeam_MuteCMD;
GVL_IO.qsTwoHandsMonitoring						:= GVL_MASTER.stSafety.bTwoHands_MonitorCMD;



// Master Machine CTRL Outputs
GVL_IO.qGripperA_Close							:= GVL_MODULES.stSmac.bGripperA_Close;
GVL_IO.qGripperA_Open							:= GVL_MODULES.stSmac.bGripperA_Open;
GVL_IO.qGripperB_Close							:= GVL_MODULES.stSmac.bGripperB_Close;
GVL_IO.qGripperB_Open							:= GVL_MODULES.stSmac.bGripperB_Open;
//GVL_IO.qCycleIndicator_GreenLED					:= GVL_MASTER.bCycleIndicator_Green;
//GVL_IO.qCycleIndicator_RedLED					:= GVL_MASTER.bCycleIndicator_Red;



// Y-Axis Outputs - 




// Kistler Outputs
GVL_IO.qControlBytes 							:= GVL_MODULES.stKistler.st_TelegramDataOut;
GVL_IO.qKistlerCTRL_Sig1						:= GVL_MODULES.stKistler.bKistlerCTRL_Sig1;
GVL_IO.qKistlerCTRL_Sig2						:= GVL_MODULES.stKistler.bKistlerCTRL_Sig2;
GVL_IO.qKistlerCTRL_Sig3						:= GVL_MODULES.stKistler.bKistlerCTRL_Sig3;
GVL_IO.qKistlerCTRL_Sig4						:= GVL_MODULES.stKistler.bKistlerCTRL_Sig4;



// Smac Outputs
GVL_IO.qGripperA_Open							:= GVL_MODULES.stSmac.bGripperA_Open;
GVL_IO.qGripperA_Close							:= GVL_MODULES.stSmac.bGripperA_Close;	
GVL_IO.qGripperB_Open							:= GVL_MODULES.stSmac.bGripperB_Open;
GVL_IO.qGripperB_Close							:= GVL_MODULES.stSmac.bGripperB_Close;

//---------------------------------------------------------------------------------------oldschoo1
END_ACTION

ACTION g_Map_StatusLamps:

// Reset Button LED Lamp
GVL_IO.qResetButton_LED := bFlash2Hz AND (stMachineStatus.bImmediateStopped OR 
								   		  stMachineStatus.bImmediateFault 	OR 
								          stMachineStatus.bCycleStopped 	OR
		   			 			          stMachineStatus.bCycleStopFault 	OR 
								          stMachineStatus.bInitialising);

		   
// Start Button LED Lamp
GVL_IO.qStartButton_LED := (stMachineStatus.bReadyToStart AND bFlash1Hz_7030) OR stMachineStatus.bAutoCycle;

(*
// Cycle Indicator LED Lamp
GVL_MASTER.bCycleIndicator_Green			:= stMachineStatus.bProcessCycle;
GVL_MASTER.bCycleIndicator_Red 				:= stMachineStatus.bAutoCycle AND NOT stMachineStatus.bProcessCycle; 
					
	*)
END_ACTION

ACTION h_Write_PersistentData:
tonWritePeristentTrig(IN := NOT bWritePersistentTrigger, 
					  PT := tWritePersistentPeriod, 
					  Q   => bWritePersistentTrigger);

fbWritePersistent(	NETID 	:= '', 
					PORT 	:= 851,
					START 	:= bWritePersistentTrigger,
					Mode 	:= E_PersistentMode.SPDM_2PASS,
					BUSY 	=> bWritePersistentBusy, 
					ERR 	=> bWritePersistentError,
					ERRID 	=> bWritePersistentErrID);
					
//----------------------------------------------------------oldschoo1
END_ACTION

ACTION i_TerminalInfo:

// TERMINAL 1 _ EK1100 - EtherCAT Coupler
GVL_IO.fbTerminalInfo[1](nTerminalState := GVL_IO.nEK1100State, 
sTerminalState => GVL_IO.sEK1100Status);
// TERMINAL 2 _ EL6070-0033	- License Key Terminal for TC3
GVL_IO.fbTerminalInfo[2](nTerminalState := GVL_IO.nEL6070State, 
sTerminalState => GVL_IO.sEL6070Status);
// TERMINAL 3 _ EL6910 - Safety PLC - Virtual Channels
GVL_IO.fbTerminalInfo[3](nTerminalState := GVL_IO.nEL6910State, 
sTerminalState => GVL_IO.sEL6910Status);
//TERMINAL 4 _ EL1918 - 8 Channel Digital Safety Inputs
GVL_IO.fbTerminalInfo[4](nTerminalState := GVL_IO.nEL1918_1State, 
sTerminalState => GVL_IO.sEL1918Status);
// TERMINAL 5 _ EL1918 - 8 Channel Digital Safety Inputs
GVL_IO.fbTerminalInfo[5](nTerminalState := GVL_IO.nEL1918_2State, 
sTerminalState => GVL_IO.sEL1918_2Status);
// TERMINAL 6 _ ELEL2904 - 4 Channel Digital Safety Outputs
GVL_IO.fbTerminalInfo[6](nTerminalState := GVL_IO.nEL2904_1State, 
sTerminalState => GVL_IO.sEL2904_1Status);
// TERMINAL 7 _ ELEL2904 - 4 Channel Digital Safety Outputs
GVL_IO.fbTerminalInfo[7](nTerminalState := GVL_IO.nEL2904_2State, 
sTerminalState => GVL_IO.sEL2904_2Status);
// TERMINAL 8 _ EL1809 - 16 Channel Digital Input Terminal
GVL_IO.fbTerminalInfo[8](nTerminalState := GVL_IO.nEL1809_1State, 
sTerminalState => GVL_IO.sEL1809_1Status);
// TERMINAL 9 _ EL1809 - 16 Channel Digital Input Terminal
GVL_IO.fbTerminalInfo[9](nTerminalState := GVL_IO.nEL1809_2State, 
sTerminalState => GVL_IO.sEL1809_2Status);
// TERMINAL 10 _ EL2809	- 16 Channel Digital Output Terminal
GVL_IO.fbTerminalInfo[10](nTerminalState := GVL_IO.nEL2809State, 
sTerminalState => GVL_IO.sEL2809Status);
// TERMINAL 11 _ EL9576 - Brake Chopper Terminal
GVL_IO.fbTerminalInfo[11](nTerminalState := GVL_IO.nEL9576State, 
sTerminalState => GVL_IO.sEL9576Status);
// TERMINAL 12 _ EL7211-0010 - Servo Motor Drive
GVL_IO.fbTerminalInfo[12](nTerminalState := GVL_IO.nEL7211State, 
sTerminalState => GVL_IO.sEL7211Status);
// BOX 13 _ maXYnos - Drive and Force Sensor for Kistler Press
GVL_IO.fbTerminalInfo[13](nTerminalState := GVL_IO.nKistlermaXYmosState, 
sTerminalState => GVL_IO.sKistlermaXYmosStatus);
END_ACTION

ACTION j_ManualMode:
IF	 GVL_MASTER.stMachineStatus.bReadyToStart THEN
	GVL_HMI.bEnableManualMode := TRUE;
ELSE GVL_HMI.bEnableManualMode := FALSE;
END_IF


GVL_HMI.rtrigManualMode(CLK:= GVL_HMI.nRegionMain=10 AND NOT GVL_HMI.rtrigManualModeOff[1].Q AND NOT GVL_HMI.rtrigManualModeOff[2].Q AND NOT GVL_HMI.rtrigManualModeOff[3].Q AND NOT GVL_HMI.rtrigManualModeOff[4].Q );
GVL_HMI.rtrigManualModeOff[1](CLK:=GVL_Master.stMachineStatus.bManualMode AND (GVL_HMI.nRegionMain <> 10));
GVL_HMI.rtrigManualModeOff[2](CLK:= rtrigStopButton.Q);
GVL_HMI.rtrigManualModeOff[3](CLK:= NOT GVL_Master.stMasterCTRL.bNoMachineImmediateFault );
GVL_HMI.rtrigManualModeOff[4](CLK := GVL_HMI.bManualModeOff[1], Q => GVL_HMI.bManualModeOff[2]);

IF GVL_HMI.rtrigManualMode.Q THEN 
	GVL_Master.stMasterCTRL.bManualModeRequest := TRUE;
	GVL_HMI.bManualModeOff[1] := FALSE;
ELSIF  GVL_HMI.rtrigManualModeOFF[1].Q OR  GVL_HMI.rtrigManualModeOFF[2].Q OR 
		GVL_HMI.rtrigManualModeOFF[3].Q THEN
		GVL_HMI.nRegionMain		:= 1;
	GVL_Master.stMasterCTRL.bManualModeRequest := FALSE ;
	GVL_HMI.bManualModeOff[1] := TRUE;
	
	
ELSE GVL_HMI.bManualModeOff[1] := FALSE;
	
END_IF
END_ACTION

END_PROGRAM

// ---- POUs/03_Utilities/FB_EventLog.TcPOU
FUNCTION_BLOCK FB_EventLog
VAR_INPUT
	bEnable				:BOOL;		//Enable alarm loggin functionality
END_VAR
VAR_IN_OUT
	sDateTime			:STRING;	//System current date and time for alarm log functinality
	aEventFlags			:ARRAY[*] OF BOOL;			//Active events array - needs to be te exact same size as aEventMsgs
	aEventTexts			:ARRAY[*] OF T_MaxSTring;	//All events messages defined for the system - indices corresponds to indices of aEvents
	aActiveEvents		:ARRAY[*] OF T_MaxSTring;	//Active events messages - displayed in active alarms
	aEventLog			:ARRAY[*] OF T_MaxSTring;	//Logged events messages - displayed in alarm history
	siDate				:STRING;	//System current Date
	siTime				:STRING;		//System current time
	soDate				:ARRAY[*] OF T_MaxSTring;
	soTime				:ARRAY[*] OF T_MaxSTring;
END_VAR
VAR_OUTPUT
	bLogActive			:BOOL;
END_VAR
VAR
	bFirstScan			:BOOL := TRUE;
	bInputDataValid		:BOOL; 	//Input data valid - checked only at first scan or block reinit
	aEventsOld			:POINTER TO BOOL;
	ni					:DINT;
	nj					:DINT;
	
	nEventsStart		:DINT;	//Start index of all arrays
	nEventsEnd			:DINT;	//End index of longest arrays - aEvents and aEventMsgs
	nEventTextsStart	:DINT;	//Start index of aEventMsgs
	nEventTextsEnd		:DINT;	//End index of aEventMsgs
	nLogEventsStart		:DINT;	//Start index of aLogEventMsgs
	nLogEventsEnd		:DINT;	//End index of aLogEventMsgs
	nActiveEventsStart	:DINT;	//Start index of aActiveEventMsgs
	nActiveEventsEnd	:DINT;	//End index of aActiveEntsMsgs
END_VAR

//Check input data
IF bFirstScan THEN
	Init();
END_IF

bLogActive := bEnable AND bInputDataValid and (aEventsOld <> 0);
IF NOT bLogActive OR (aEventsOld = 0) THEN
	RETURN; //Do nothing
END_IF

//Update active and logged events
IF EventChangeDetected() THEN
	//Update event log
	FOR ni := nEventsEnd TO nEventsStart BY -1 DO
		
		//Check for new active alarms
		IF aEventFlags[ni] AND NOT aEventsOld[ni] THEN
			//Shift all alarms one row down
			FOR nj := nLogEventsEnd TO nLogEventsStart + 1 BY -1 DO
				aEventLog[nj] := aEventLog[nj-1];
				soDate	[nj]	:= soDate[nj-1];
				soTime	[nj]	:= soTime[nj-1];
			END_FOR
			
			//Add new logged event
			aEventLog[nEventsStart] := aEventTexts[ni];
			soDate	[nEventsStart]	:= siDate;
			soTime	[nEventsStart]	:= siTime;
		END_IF
	END_FOR
	
	//Clear all active event messages initially
	ClearActiveMsgs();
	
	//Update active events
	ni := nEventsStart;
	nj := nActiveEventsStart;
	WHILE ni <= nEventsEnd AND nj <= nActiveEventsEnd DO
		IF aEventFlags[ni] THEN //If Alarm is active, move the corresponding Alarm Message into the IntermediateAlarmTable
			aActiveEvents[nj] := aEventTexts[ni];
			nj := nj+1;
		END_IF
		ni := ni+1;
	END_WHILE
	
	//Update aEventsOld for comparison
	StoreEvents();
END_IF

bFirstScan := FALSE;

//Calculate bounds for all arrays
METHOD PRIVATE CalcBounds : BOOL
VAR_INPUT
END_VAR
//Calculate indices for all arrays
nEventsStart := LOWER_BOUND(aEventFlags, 1);
nEventsEnd := UPPER_BOUND(aEventFlags, 1);
nEventTextsStart := LOWER_BOUND(aEventTexts, 1);
nEventTextsEnd := UPPER_BOUND(aEventTexts, 1);
nLogEventsStart := LOWER_BOUND(aEventLog, 1);
nLogEventsEnd := UPPER_BOUND(aEventLog, 1);
nActiveEventsStart := LOWER_BOUND(aActiveEvents, 1);
nActiveEventsEnd := UPPER_BOUND(aActiveEvents, 1);
END_METHOD

//Clear active messages on events update
METHOD PRIVATE ClearActiveMsgs : BOOL
VAR
	ni		:DINT;
END_VAR
//Clear active messages one-by-one
FOR ni := nActiveEventsStart TO nActiveEventsEnd DO
	aActiveEvents[ni] := '';
END_FOR
END_METHOD

//Event change detected
METHOD PRIVATE EventChangeDetected : BOOL
VAR
	ni			:DINT;
	nj			:DINT;
END_VAR
//Compare events change one-by-one to dynamic array
EventChangeDetected := FALSE;
nj := 0; //Index for aEventsOld array

FOR ni := nEventsStart TO nEventsEnd DO
	IF aEventFlags[ni] <> aEventsOld[nj] THEN
		EventChangeDetected := TRUE;	
		RETURN;
	END_IF
	nj := nj + 1;
END_FOR
END_METHOD

METHOD FB_exit : BOOL
VAR_INPUT
	bInCopyCode : BOOL; // if TRUE, the exit method is called for exiting an instance that is copied afterwards (online change).
END_VAR
//Clear dynamically allocated data on block close
IF aEventsOld <> 0 THEN
	__DELETE(aEventsOld);
END_IF
END_METHOD

METHOD PRIVATE Init : BOOL
VAR_INPUT
END_VAR
//Calculate bounds for all referenced arrays
CalcBounds();
bInputDataValid := InputDataValid();

//Check if dynamic array creted
IF bInputDataValid AND aEventsOld = 0 THEN
	aEventsOld := __NEW(BOOL, TO_UDINT(nEventsEnd - nEventsStart + 1));
END_IF
END_METHOD

METHOD PRIVATE InputDataValid : BOOL
VAR_INPUT
END_VAR
InputDataValid := nEventsStart = nEventTextsStart AND nEventsEnd = nEventTextsEnd;
END_METHOD

//Store previous events in aEventsOld
METHOD PRIVATE StoreEvents : BOOL
VAR
	ni		:DINT;
	nj		:DINT;
END_VAR
//Copy one-by-one elements from aEvents to aEventsOld
nj := 0; //Index for aEventsOld array
FOR ni := nEventsStart TO nEventsEnd DO
	aEventsOld[nj] := aEventFlags[ni];
	nj := nj + 1;
END_FOR

StoreEvents := TRUE;
END_METHOD

END_FUNCTION_BLOCK

// ---- POUs/00_MASTER/PRG_MasterSystemTime.TcPOU
PROGRAM PRG_MasterSystemTime
VAR
		//Variables
	bReadyToRead				:BOOL;
	bFirstScan					:BOOL := TRUE;
	bUpdateSysTime				:BOOL; //Output of pulse generator
	tSysTimeUpdatePeriod		:TIME := T#5S;
	stTimeStamp					:TIMESTRUCT;
	stNullTimeStamp				:TIMESTRUCT;
	sRawDateTime				:STRING;
	sSystemDate					:STRING;
	sSystemTime					:STRING;
	sDateTime					:STRING;
	sDateTimeSpaces				:STRING;
	
	stTimeTest                  :TIMESTRUCT;
	sttimeTest2                 :TIMESTRUCT;
	sTestTime                   :STRING;
	nSectTest                   :DINT;
	bStartTest                  :BOOL;
	bStsrtTest2                 :BOOL;
	
	
	//Functions
	fbGetSystemTime				:TC2_Utilities.NT_GetTime;
	fbRTClock					:TC2_Utilities.RTC_EX2;		//Local real-time clock
	tonTimeUpdateGen			:TC2_Utilities.TON;			//Pulse generator for triggering fbGetSystemTime function
	rtrigSysTimeCollected		:TC2_Utilities.R_TRIG;		//System time collected

    fbTimerControl              :FB_TimeControl;
	bStartTimeTest              :BOOL;
	bResetTimeTest              :BOOL;
	nTimeHourTest               :DINT;
	nTimeMinTest                :DINT;
	nTimeSecTest                :DINT;
	nTimeTotalSecTest           :DINT;
END_VAR

//Aux functions call
tonTimeUpdateGen(	IN := NOT bUpdateSysTime,
					PT := tSysTimeUpdatePeriod,
					Q => bUpdateSysTime);

//bReadyToRead :=  Tc2_System.MEMCMP( ADR( stTimeStamp), ADR (stNullTimeStamp), SIZEOF(stTimeStamp)) <> 0 AND NOT  fbGetSystemTime.BUSY;	
			(*keczi*)	(*zrobione po to zeby w wypadku jak po starcie PLC na HMI mial pokazywac czas alarmu '00:00:00', zebyb poczekal az faktycznie pokazuje date i czas*)

//Get Current System Time
fbGetSystemTime(NETID := ,
				START := bFirstScan OR bUpdateSysTime,
				TMOUT := ,
				BUSY => ,
				ERR => ,
				ERRID => ,
				TIMESTR => );
				
//Get system time done detection - one-shot
rtrigSysTimeCollected(CLK := NOT fbGetSystemTime.BUSY);

//Synchronize Real-Time clock with system time
fbRTClock(	EN := rtrigSysTimeCollected.Q, 
			PDT := fbGetSystemTime.TIMESTR,
			CDT => stTimeStamp, 
			Q => bReadyToRead);

// System Date and Time in Proper Order 
IF bReadyToRead THEN
	sRawDateTime := SYSTEMTIME_TO_STRING(stTimeStamp);  // format: YYYY-MM-DD-hh:mm:ss.xxx
	sSystemDate := CONCAT(CONCAT(CONCAT(CONCAT(MID(sRawDateTime, 2, 9), '.'),  MID(sRawDateTime, 2, 6)), '.'), LEFT(sRawDateTime, 4));
	sSystemTime := MID(sRawDateTime, 8, 12);
	sDateTime := CONCAT(CONCAT(sSystemDate, '  '), sSystemTime);
	sDateTimeSpaces	:= CONCAT(sDateTime, '    ');
	
	//Time to write to CSV Files
	//nSystemTime := sSystemTime;
END_IF;

bFirstScan := FALSE;

IF bStartTest THEN
	sTestTime:= SYSTEMTIME_TO_STRING(stTimeTest);
END_IF

fbTimerControl( bEnable  :=  bStartTimeTest,
	            bReset   :=  bResetTimeTest,
				nHour     => nTimeHourTest,
				nMin      => nTimeMinTest,
				nSec      => nTimeSecTest,
				nTotalSec => nTimeTotalSecTest );

GVL_MASTER.sSystemDate 		:= sSystemDate;
GVL_MASTER.sSystemTime		:= sSystemTime;

END_PROGRAM

// ---- POUs/03_Utilities/FB_TimeControl.TcPOU
FUNCTION_BLOCK PUBLIC FB_TimeControl
VAR_INPUT
	bEnable         :BOOL;
	bReset          :BOOL;
END_VAR
VAR_OUTPUT 
	nHour           :DINT;
	nMin            :DINT;
	nSec            :DINT;
	nTotalSec       :DINT;
END_VAR
VAR
	tpPulse1        :TP;
	tpPulse2        :TP;
	
	
    bMainStart      :BOOL;
    bStart1         :BOOL;
    bStart2         :BOOL;
    bStop           :BOOL;
    bPuls1          :BOOL;
    bPuls2          :BOOL;

    ftrigPuls1      :F_TRIG;
    ftrigPuls2      :F_TRIG;
    rtrigPulsMain   :R_TRIG;
	
	
END_VAR

rtrigPulsMain(CLK:= bEnable);
ftrigPuls1(CLK:= bPuls2);
ftrigPuls2(CLK:= bPuls1);

tpPulse1(IN:=(ftrigPuls1.Q OR rtrigPulsMain.Q) ,PT:= T#490MS);
bPuls1:= tpPulse1.Q;

tpPulse2(IN:=(ftrigPuls2.Q AND NOT bStop) ,PT:= T#490MS);
bPuls2:=tpPulse2.Q;

IF bEnable THEN
	bMainStart := TRUE;
ELSE 
	bMainStart := FALSE;
END_IF
bStop := NOT bMainStart;

IF bMainStart AND ftrigPuls1.Q THEN
	nTotalSec := nTotalSec + 1;
ELSIF bReset THEN
	nTotalSec := 0;
END_IF
//Secend
IF bMainStart AND ftrigPuls1.Q THEN
	nSec := nSec + 1;
	ELSIF (nSec = 60) THEN
	nSec := 0;
	ELSIF bReset THEN
	nSec := 0;	
END_IF
//Minutes
IF bMainStart THEN
	nMin := (nTotalSec-(nHour*3600)) /60;
	ELSIF bReset THEN
	nMin := 0;
END_IF
//Hours
IF bMainStart THEN
	nHour := nTotalSec/3600;
	ELSIF bReset THEN
	nHour := 0;
END_IF

END_FUNCTION_BLOCK

// ---- POUs/01_MODULES/AXIS_Y/Y_Master_Y_Axis.TcPOU
PROGRAM Y_Master_Y_Axis
VAR
	
	// Link to Task
	refY_Axis							:AXIS_REF;	//Axis_1
										
										
	fPositionLimitMin					:LREAL			 := 5;
	fPositionLimitMax					:LREAL			 := 110;
	fLimitPositionLow					:LREAL; 		//16#0001_000D
	fLimitPositionHigh					:LREAL;			//16#0001_000E
	
	// Local Axis Config
	posTarget							:LREAL;
	fOffsets							:ARRAY [1..3]OF LREAL;
	nOfSetPos							:INT:=3;
	fCurrentPosition					:LREAL;

    // State Machine CTRL
    eState								:E_AxisState:=E_AxisState.ABORTED;

	// Timers && Triggers
	tonResetError						:Tc2_Standard.TON;
	tonPowerAxis						:Tc2_Standard.TON;
	tonPowerAxis2						:Tc2_Standard.TON;
	tonActionDone						:Tc2_Standard.TON;
	tonMoveTimeout						:Tc2_Standard.TON;
	tonPowerUpTimeout					:Tc2_Standard.TON;
	tonPowerUpError						:Tc2_Standard.TON;
	tonAbortModule						:Tc2_Standard.TON;
	tonDelayExe							:Tc2_Standard.TON;

				
    // Motion FB Instances
    fbPower    							:Tc2_MC2.MC_Power;
    fbReset    							:Tc2_MC2.MC_Reset;
    fbStop     							:Tc2_MC2.MC_Stop;
    fbMoveABS     						:Tc2_MC2.MC_MoveAbsolute;
	fbMoveREL							:Tc2_MC2.MC_MoveRelative;
	fbReadStatus						:Tc2_MC2.MC_ReadStatus;
	fbReadPos							:Tc2_MC2.MC_ReadActualPosition;
	stAxisStatus						:ST_AxisStatus;
	fbParameter							:ARRAY[0..1]OF Tc2_MC2.MC_ReadParameter;
	
	// Function Blocks Flags
	bReq_Power							:BOOL;		// Request Power to Axis 
	bReq_Reset							:BOOL;		// Request Axis Reset
	bReq_MoveABS						:BOOL;		// Request Move Action 
	bReq_MoveREL						:BOOL;		// Request Move Action
	bReq_Stop							:BOOL;		// Request Axis to Stop
	bAxisInError						:BOOL;
	
	//Index
	idx									:INT;
	//MANUAL MODE
	nManualModeState					:DINT;
	trigbMoveToPos						:R_TRIG;
	bTest								:BOOL;

//-------------------------------------------------------------------------------*		
END_VAR
VAR_INPUT	
	bRetract							:BOOL;		// Velocity Change
END_VAR
VAR PERSISTENT
		// Set Parameters
    cfgAxis    							:ST_Y_Axis;(*:=(
										posHome 		  := 7.0,
										posWorkPositions := [14.5,33.7,100.0],
										fPositionOffsets := [0.0,  0.0,  0.0],
										fTargetVelocity  := 25.0,
										fRetractVelocity := 90.0);//after comes from hmi*)
END_VAR

//--------------------IN/OUT-----------------------------------------------------*
VAR_INPUT	
	CMD									:ST_ModuleCMD;	
END_VAR
VAR_OUTPUT	
	STATUS								:ST_ModuleStatus;	
END_VAR
//------------------------------------------------------------------------oldschoo1

PRG_Fault_Axis_Y(aAlarms := GVL_Master.stAlarms);
// Positions Offsets Mapping
IF (GVL_PERSISTENT.fPositions_Offset[1]>1.3) OR (GVL_PERSISTENT.fPositions_Offset[2]>1.3)
	THEN
fOffsets[1] := 0.0;
fOffsets[2] := 0.0;
ELSE
fOffsets[1] := GVL_PERSISTENT.fPositions_Offset[1];	//Picking Screw Position
fOffsets[2] := GVL_PERSISTENT.fPositions_Offset[2];	//Screwwing and Pressing Actions Position	
END_IF

//-------------------------------------------------------------------------------------------*
//Call For Actions
a_Ctrl_Axis();
b_Call_AxisFBs();
d_Get_CurrentPosition();
//---------------------*
//------------------------------------------------------------------------------------oldschoo1

ACTION a_Ctrl_Axis:
// Timmers && Triggers     
tonPowerAxis	(IN:= eState=E_AxisState.ENABLE_POWER, 
			 	 PT:= T#50MS);			 
tonActionDone	(IN:= eState=E_AxisState.IN_TARGET_POS,
			  	 PT:= T#100MS);
tonMoveTimeout	(IN:= eState=E_AxisState.MOVE_ABS OR eState=E_AxisState.MOVE_REL,
			   	 PT:= T#10S);			  
tonAbortModule	(IN:=	cmd.bAbort OR (NOT stSafety.bSafety_OK) OR (NOT cmd.bEnable),
			     PT:= T#100MS);
tonResetError	(IN:= cmd.bReset OR fbPower.Error OR fbStop.Error OR fbMoveABS.Error OR fbMoveREL.Error,
			  	 PT:= T#500MS);
tonDelayExe  	(IN:= eState=E_AxisState.HOMING AND stY_Axis.bSetToHome,
			  	 PT:= T#300MS);
(**************************************************RESET************************************************)		   
// Reset Errors
IF cmd.bReset OR fbPower.Error OR fbStop.Error OR fbMoveABS.Error OR fbMoveREL.Error THEN

			status.bError 	:= TRUE;
			bReq_Power 		:= FALSE;
			bReq_MoveABS 	:= FALSE;
			bReq_MoveREL 	:= FALSE;
			bReq_Stop 		:= FALSE;		
            eState := E_AxisState.RESET_ERROR;
			END_IF
IF  eState=E_AxisState.ABORTED THEN
CMD_Axis.bExecute			  :=FALSE;
stY_Axis.bSetToHome			  :=FALSE;
Y_Master_Y_Axis.bRetract 	  :=FALSE; END_IF			
IF tonResetError.Q THEN bReq_Reset := TRUE; END_IF
IF bAxisInError THEN bReq_Reset:=bResetButtonRisingEdge; eState:= E_AxisState.ERROR; END_IF

// Abort Action
IF tonAbortModule.Q THEN

			bReq_Power := FALSE;
			eState := E_AxisState.ABORTED;
			END_IF
IF CMD.bManualMode THEN
	eState := E_AxisState.MANUAL_MODE;
END_IF
(*******************************************************CTRL***********************************************************)
// Axis CTRL State Machine
CASE eState OF //--------------------------------------------------------------------------------------------------SM
	
E_AxisState.ABORTED://-------------------------------------------------------------------------------------------ABORTED:


							IF stSafety.bSafety_OK AND cmd.bEnable AND NOT fbPower.Error THEN
								
									bReq_Power := TRUE;
									eState := E_AxisState.ENABLE_POWER;
							END_IF

E_AxisState.ENABLE_POWER://---------------------------------------------------------------------------------ENABLE_POWER:

							IF fbPower.Status AND NOT fbPower.Error THEN
								
									bReq_Reset := TRUE;
									eState := E_AxisState.HOMING;
							END_IF

E_AxisState.RESET_ERROR://-----------------------------------------------------------------------------------RESET_ERROR:

							IF fbReset.Done AND fbPower.Status THEN
								
									bReq_Reset := FALSE;
									eState := E_AxisState.HOMING;
									
							ELSIF fbReset.Done AND NOT fbPower.Status THEN
							
										eState := E_AxisState.ABORTED;
										
							ELSIF NOT fbPower.Error AND NOT fbStop.Error AND 
								  NOT fbMoveABS.Error AND NOT fbMoveREL.Error THEN
								  
										eState := E_AxisState.ABORTED;
							END_IF

E_AxisState.HOMING://---------------------------------------------------------------------------------------------HOMING:

							IF ABS(fCurrentPosition - cfgAxis.posHome)<=0.5 THEN
								
										bReq_MoveABS				  :=FALSE;
										CMD_Axis.bExecute			  :=FALSE;
										stY_Axis.bSetToHome			  :=FALSE;
										Y_Master_Y_Axis.bRetract 	  :=FALSE;
										
										eState := E_AxisState.AXIS_READY;	
 							ELSE
										//bReq_MoveABS				  :=TRUE; //test
										stY_Axis.bSetToHome			  :=TRUE;
										posTarget:=cfgAxis.posHome;
										Y_Master_Y_Axis.bRetract 	  :=TRUE;
										eState 							:= E_AxisState.MOVE_ABS;
							END_IF
							 	
									IF tonDelayExe.Q THEN
											CMD_Axis.bExecute		  :=TRUE;
									END_IF
									
E_AxisState.AXIS_READY://-------------------------------------------------------------------------------------AXIS_READY:

							IF cmd.bExecute THEN
									eState := E_AxisState.GET_TARGET;
							END_IF
							
E_AxisState.GET_TARGET://-------------------------------------------------------------------------------------GET_TARGET:

							posTarget := c_Get_TargetPositon(
															posHome 	:= cfgAxis.posHome,
															posPoints   := cfgAxis.posWorkPositions,
															fOffsets	:= fOffsets,
															bSetHome 	:= stY_Axis.bSetToHome,
															bSetPoint 	:= stY_Axis.bSetToPosition
															);	
															eState := E_AxisState.MOVE_ABS;
	
